(*FB_Init is always available implicitly and it is used primarily for initialization.
The return value is not evaluated. For a specific influence, you can also declare the
methods explicitly and provide additional code there with the standard initialization
code. You can evaluate the return value.*)
METHOD FB_Init : BOOL
VAR_INPUT
	(* TRUE: the retain variables are initialized (reset warm / reset cold)*)
	bInitRetains : BOOL;

	(* TRUE: the instance will be copied to the copy code afterward (online change)   *)
	bInCopyCode : BOOL;
	Name		: T_MaxString;
	Cylinder	: I_Cylinder;
END_VAR
THIS^.Cylinder := Cylinder;
Events.GenerateTcEvents(Cylinder.Name, ADR(TC_events.Cylinder), SIZEOF(ST_Cylinder));
END_METHOD

END_FUNCTION_BLOCK

// Events/Interface/I_EventReactionTcEvents
INTERFACE I_EventReactionTcEvents EXTENDS I_EventReaction

METHOD GetHighestActiveEventSeverity : TcEventSeverity
END_METHOD

END_INTERFACE

// Events/Interface/I_EventReaction
INTERFACE I_EventReaction EXTENDS I_Resettable

METHOD GetHighestActiveEventReaction : DINT;
END_METHOD

METHOD SetEventReactions
VAR_INPUT
	Verbose	 : DINT := 0;
	Info	 : DINT := 1;
	Warning	 : DINT := 2;
	Error	 : DINT := 3;
	Critical : DINT := 4;
END_VAR
END_METHOD

END_INTERFACE

// Events/TcEventClass
{attribute 'enable_dynamic_creation'}
FUNCTION_BLOCK TcEventClass EXTENDS CyclicComponent IMPLEMENTS I_EventClassTcEvents
VAR
	pEventClass				   : PVOID;
	pEventBuffer			   : POINTER TO PVOID;
	pEventTriggerBuffer		   : POINTER TO PVOID;
	pEventAutoResetBuffer	   : POINTER TO PVOID;
	NullEvent				   : FB_TcAlarm;
	NullBool				   : BOOL;
	NumberOfEvents			   : UDINT;
	HighestActiveEventSeverity : TcEventSeverity;
	EventReactionVerbose	   : DINT := 0;
	EventReactionInfo		   : DINT := 1;
	EventReactionWarning	   : DINT := 2;
	EventReactionError		   : DINT := 3;
	EventReactionCritical	   : DINT := 4;
	TcEventClassArguments	   : TcEventClassArguments;
END_VAR

METHOD Dispose
VAR
	i				: UDINT;
	pEvent			: POINTER TO FB_TcAlarm;
	pDispose		: POINTER TO TcEventClass;
	pEventAutoReset : POINTER TO BOOL;
END_VAR
pDispose := THIS;
FOR i := 1 TO NumberOfEvents DO
	pEvent := GetEventInstance(i);
	__DELETE(pEvent);
	pEventAutoReset := GetEventAutoResetInstance(i);
	__DELETE(pEventAutoReset);
END_FOR

__DELETE(pEventBuffer);
__DELETE(pDispose);
__DELETE(pEventTriggerBuffer);
__DELETE(pEventAutoResetBuffer);
END_METHOD

//FB_Exit must be implemented explicitly. If there is an implementation, then the

//method is called before the controller removes the code of the function block instance

//(implicit call). The return value is not evaluated.
METHOD FB_Exit : BOOL
VAR_INPUT
	bInCopyCode : BOOL; // TRUE: the exit method is called in order to leave the instance which will be copied afterwards (online change).  
END_VAR

VAR
	i				: UDINT;
	pEvent			: POINTER TO FB_TcAlarm;
	pEventAutoReset : POINTER TO BOOL;
END_VAR
FOR i := 1 TO NumberOfEvents DO
	pEvent := GetEventInstance(i);
	__DELETE(pEvent);
	pEventAutoReset := GetEventAutoResetInstance(i);
	__DELETE(pEventAutoReset);
END_FOR

__DELETE(pEventBuffer);
__DELETE(pEventTriggerBuffer);
__DELETE(pEventAutoResetBuffer);
END_METHOD

METHOD ClearEventById
VAR_INPUT
	EventId : UDINT;
END_VAR

VAR
	pEvent : POINTER TO FB_TcAlarm;
END_VAR
IF CheckEventId(EventId) THEN
	pEvent := GetEventInstance(EventId);
	IF (pEvent <> 0) THEN
		IF pEvent^.bRaised THEN
			pEvent^.Clear();
			FindActiveSeverity();
		END_IF
	END_IF
END_IF
END_METHOD

METHOD GetHighestActiveEventReaction : DINT
CASE HighestActiveEventSeverity OF
	TcEventSeverity.Verbose:
		GetHighestActiveEventReaction := EventReactionVerbose;

	TcEventSeverity.Info:
		GetHighestActiveEventReaction := EventReactionInfo;

	TcEventSeverity.Warning:
		GetHighestActiveEventReaction := EventReactionWarning;

	TcEventSeverity.Error:
		GetHighestActiveEventReaction := EventReactionError;

	TcEventSeverity.Critical:
		GetHighestActiveEventReaction := EventReactionCritical;
END_CASE
END_METHOD

METHOD GetHighestActiveEventSeverity : TcEventSeverity
GetHighestActiveEventSeverity := HighestActiveEventSeverity;
END_METHOD

{attribute 'monitoring' := 'call'}
PROPERTY IsResettable : BOOL
GET
VAR
	i		  : UDINT;
	pEvent	  : POINTER TO FB_TcAlarm;
	pTrigger  : POINTER TO BOOL;
END_VAR
IsResettable := FALSE;
FOR i := 1 TO NumberOfEvents DO
	pTrigger := GetEventTriggerInstance(i);
	IF (pTrigger <> 0) THEN
		pEvent := GetEventInstance(i);
		IF (pEvent <> 0) AND_THEN NOT pTrigger^ AND pEvent^.bRaised THEN
			IsResettable := TRUE;
		END_IF
	END_IF
END_FOR
END_GET
END_PROPERTY

METHOD RaiseEvent
VAR_INPUT
	EventId	  : UDINT;
END_VAR

VAR
	pEvent : POINTER TO FB_TcAlarm;
END_VAR
IF CheckEventId(EventId) THEN
	pEvent := GetEventInstance(EventId);
	IF (pEvent <> 0) THEN
		IF NOT pEvent^.bRaised THEN
			pEvent^.Raise();
			IF pEvent^.eSeverity > HighestActiveEventSeverity THEN
				HighestActiveEventSeverity := pEvent^.eSeverity;
			END_IF

			pEvent^.ipArguments.Clear();
		END_IF
	END_IF
END_IF
END_METHOD

METHOD ResetBySeverity : BOOL
VAR_INPUT
	Severity : UDINT;
END_VAR

VAR
	i	   : UDINT;
	pEvent : POINTER TO FB_TcAlarm;
END_VAR
FOR i := 1 TO NumberOfEvents DO
	pEvent := GetEventInstance(i);
	IF (pEvent <> 0) AND_THEN (pEvent^.eSeverity <= TO_DINT(Severity)) THEN
		pEvent^.Clear();
	END_IF
END_FOR

FindActiveSeverity();
ResetBySeverity := TRUE;
END_METHOD

METHOD SetEvent
VAR_INPUT
	EventId	  : UDINT;
	Trigger	  : POINTER TO BOOL;
	AutoReset : BOOL;
END_VAR

VAR
	pBool : POINTER TO BOOL;
END_VAR
IF CheckEventId(EventId) THEN
	IF Trigger <> 0 THEN
		SetEventTriggerInstance(EventId, Trigger);
	END_IF

	pBool  := GetEventAutoResetInstance(EventId);
	pBool^ := AutoReset;
END_IF
END_METHOD

METHOD SetEventReactions
VAR_INPUT
	Verbose	 : DINT := 0;
	Info	 : DINT := 1;
	Warning	 : DINT := 2;
	Error	 : DINT := 3;
	Critical : DINT := 4;
END_VAR
EventReactionVerbose  := Verbose;
EventReactionInfo	  := Info;
EventReactionWarning  := Warning;
EventReactionError	  := Error;
EventReactionCritical := Critical;
END_METHOD

METHOD PROTECTED CheckEventId : BOOL
VAR_INPUT
	EventId : UDINT;
END_VAR
CheckEventId := (EventID > 0) AND (EventId <= NumberOfEvents) AND (pEventBuffer <> 0);
END_METHOD

METHOD PROTECTED FindActiveSeverity
VAR
	i	   : UDINT;
	pEvent : POINTER TO FB_TcAlarm;
END_VAR
HighestActiveEventSeverity := Global.TcEventSeverity.Verbose;
FOR i := 1 TO NumberOfEvents DO
	pEvent := GetEventInstance(i);
	IF (pEvent <> 0) AND_THEN pEvent^.bRaised AND_THEN pEvent^.eSeverity > HighestActiveEventSeverity THEN
		HighestActiveEventSeverity := pEvent^.eSeverity;
	END_IF
END_FOR
END_METHOD

METHOD PROTECTED GetEventAutoResetInstance : POINTER TO BOOL
VAR_INPUT
	EventId : UDINT;
END_VAR

VAR
	ppEventAutoReset : POINTER TO POINTER TO BOOL;
END_VAR
IF CheckEventId(EventId) THEN
	ppEventAutoReset := pEventAutoResetBuffer + ((EventId - 1) * SIZEOF(PVOID));
	GetEventAutoResetInstance := ppEventAutoReset^;
ELSE
	GetEventAutoResetInstance := ADR(NullBool);
END_IF
END_METHOD

METHOD PROTECTED GetEventInstance : POINTER TO FB_TcAlarm
VAR_INPUT
	EventId : UDINT;
END_VAR

VAR
	ppEvent : POINTER TO POINTER TO FB_TcAlarm;
END_VAR
IF CheckEventId(EventId) THEN
	ppEvent			 := pEventBuffer + ((EventId - 1) * SIZEOF(PVOID));
	GetEventInstance := ppEvent^;
ELSE
	GetEventInstance := ADR(NullEvent);
END_IF
END_METHOD

METHOD PROTECTED GetEventTriggerInstance : POINTER TO BOOL
VAR_INPUT
	EventId : UDINT;
END_VAR

VAR
	ppEventTrigger : POINTER TO POINTER TO BOOL;
END_VAR
IF CheckEventId(EventId) THEN
	ppEventTrigger := pEventTriggerBuffer + ((EventId - 1) * SIZEOF(PVOID));
	GetEventTriggerInstance := ppEventTrigger^;
ELSE
	GetEventTriggerInstance := ADR(NullBool);
END_IF
END_METHOD

METHOD PROTECTED SetEventTriggerInstance
VAR_INPUT
	EventId : UDINT;
    Trigger : POINTER TO BOOL;
END_VAR

VAR
	ppEventTrigger : POINTER TO POINTER TO BOOL;
END_VAR
IF CheckEventId(EventId) THEN
	ppEventTrigger	:= pEventTriggerBuffer + ((EventId - 1) * SIZEOF(PVOID));
	ppEventTrigger^ := Trigger;
END_IF
END_METHOD

METHOD Reset
VAR
	i		 : UDINT;
	pEvent	 : POINTER TO FB_TcAlarm;
	pTrigger : POINTER TO BOOL;
END_VAR
FOR i := 1 TO NumberOfEvents DO
	pTrigger := GetEventTriggerInstance(i);
	pEvent	 := GetEventInstance(i);
	IF (pEvent <> 0) THEN
		IF (pTrigger <> 0) AND_THEN NOT pTrigger^ THEN
			pEvent^.Clear();
		END_IF

		IF (pTrigger = 0) THEN
			pEvent^.Clear();
		END_IF
	END_IF
END_FOR

HighestActiveEventSeverity := Global.TcEventSeverity.Verbose;
END_METHOD

METHOD PUBLIC Arguments : I_EventArguments
VAR_INPUT
	EventId : UDINT;
END_VAR

VAR
	pEvent : POINTER TO FB_TcAlarm;
END_VAR
IF CheckEventId(EventId) THEN
	pEvent := GetEventInstance(EventId);
	IF (pEvent <> 0) THEN
		TcEventClassArguments.Event := pEvent;
	ELSE
		TcEventClassArguments.Event := ADR(NullEvent);
	END_IF
ELSE
	TcEventClassArguments.Event := ADR(NullEvent);
END_IF

Arguments := TcEventClassArguments;
END_METHOD

METHOD CyclicLogic
VAR
	i	   : UDINT;
	pEvent : POINTER TO FB_TcAlarm;
	pTrigger  : POINTER TO BOOL;
    AutoReset : BOOL;
END_VAR
FOR i := 1 TO NumberOfEvents DO
	pTrigger := GetEventTriggerInstance(i);
	IF (pTrigger <> 0) THEN
		pEvent	  := GetEventInstance(i);
		AutoReset := GetEventAutoResetInstance(i)^;
		IF (pEvent <> 0) AND_THEN AutoReset AND NOT pTrigger^ THEN
			pEvent^.Clear();
			FindActiveSeverity();
		END_IF

		IF (pEvent <> 0) AND_THEN pTrigger^ THEN
			pEvent^.Raise(0);
			FindActiveSeverity();
		END_IF
	END_IF
END_FOR
END_METHOD

METHOD PUBLIC GenerateTcEvents
VAR_INPUT
	Name   : T_MaxString;
	pClass : PVOID; // ADR(TC_Events.XY) - TC Event Class in TypeSystem
	nSize  : UDINT; // SIZEOF(ST_XY) - TC Event Class in TypeSystem
END_VAR

VAR
	i				 : UDINT;
	pEventDef		 : POINTER TO TcEventEntry;
	pEvent			 : POINTER TO FB_TcAlarm;
	pBuffer			 : PVOID;
	ppBuffer		 : POINTER TO POINTER TO FB_TcAlarm;
	SourceInfo		 : FB_TcSourceInfo;
	pEventAutoReset	 : POINTER TO BOOL;
	ppEventAutoReset : POINTER TO POINTER TO BOOL;
END_VAR
NumberOfEvents		  := nSize / SIZEOF(TcEventEntry);
pEventBuffer		  := __NEW(PVOID, NumberOfEvents);
pEventTriggerBuffer	  := __NEW(PVOID, NumberOfEvents);
pEventAutoResetBuffer := __NEW(PVOID, NumberOfEvents);
pEventClass			  := pClass;
IF pEventBuffer <> 0 THEN
	SourceInfo.ResetToDefault();
	SourceInfo.sName := Name;
	FOR i := 1 TO NumberOfEvents DO
		pEvent	  := __NEW(FB_TcAlarm);
		ppBuffer  := pEventBuffer + ((i - 1) * SIZEOF(PVOID));
		ppBuffer^ := pEvent;
		pEventDef := pEventClass + ((i - 1) * SIZEOF(TcEventEntry));
		pEvent^.CreateEx2(pEventDef^, SourceInfo);

		//
		pEventAutoReset	  := __NEW(BOOL);
		ppEventAutoReset  := pEventAutoResetBuffer + ((i - 1) * SIZEOF(PVOID));
		ppEventAutoReset^ := pEventAutoReset;
	END_FOR
END_IF
END_METHOD

END_FUNCTION_BLOCK

// Events/Interface/I_EventClassTcEvents
INTERFACE I_EventClassTcEvents EXTENDS I_EventClass

METHOD PUBLIC GenerateTcEvents
VAR_INPUT
	Name   : T_MaxString;
	pClass : PVOID; // ADR(TC_Events.XY) - TC Event Class in TypeSystem
	nSize  : UDINT; // SIZEOF(ST_XY) - TC Event Class in TypeSystem
END_VAR
END_METHOD

METHOD GetHighestActiveEventSeverity : TcEventSeverity
END_METHOD

END_INTERFACE

// Events/Interface/I_EventClass
INTERFACE I_EventClass EXTENDS I_EventReaction, I_Resettable

METHOD PUBLIC Arguments : I_EventArguments
VAR_INPUT
	EventId : UDINT;
END_VAR
END_METHOD

METHOD PUBLIC ClearEventById
VAR_INPUT
	EventId : UDINT;
END_VAR
END_METHOD

{attribute 'monitoring' := 'call'}
PROPERTY IsResettable : BOOL
GET
END_GET
END_PROPERTY

METHOD PUBLIC RaiseEvent
VAR_INPUT
	EventId	  : UDINT;
END_VAR
END_METHOD

METHOD ResetBySeverity : BOOL
VAR_INPUT
	Severity : UDINT;
END_VAR
END_METHOD

METHOD SetEvent
VAR_INPUT
	EventId	  : UDINT;
	Trigger	  : POINTER TO BOOL;
	AutoReset : BOOL;
END_VAR
END_METHOD

END_INTERFACE

// Components/Digital/Visitor/ForceVisitor
FUNCTION_BLOCK ForceVisitor IMPLEMENTS I_ComponentVisitor
VAR
	Forcible : I_ForcibleBool;
	{attribute 'hide'}
	_ForceState : E_ForceState;
END_VAR

{attribute 'monitoring' := 'call'}
PROPERTY Force : E_ForceState
GET
Force := _ForceState;
END_GET
SET
_ForceState := Force;
END_SET
END_PROPERTY

METHOD VisitComponent
VAR_INPUT
	Component : I_Component;
END_VAR
IF __QUERYINTERFACE(Component, Forcible) THEN
	Forcible.Force := Force;
END_IF
END_METHOD

END_FUNCTION_BLOCK

// Components/Digital/Visitor/ReleaseAllForceVisitor
FUNCTION_BLOCK ReleaseAllForceVisitor IMPLEMENTS I_ModuleVisitor, I_ComponentVisitor
VAR
END_VAR

METHOD ReleaseForces : BOOL;
VAR_INPUT
	Module : I_Module;
END_VAR
Module.Accept(THIS^);
END_METHOD

METHOD VisitComponent
VAR_INPUT
	Component : I_Component;
END_VAR

VAR_INST
	Forcible : I_ForcibleBool;
END_VAR
IF __QUERYINTERFACE(Component, Forcible) THEN
	Forcible.Force := E_ForceState.Unforced;
END_IF
END_METHOD

METHOD VisitModule
VAR_INPUT
	Module : I_Module;
END_VAR
Module.Components.Accept(THIS^);
Module.Modules.Accept(THIS^);
END_METHOD

END_FUNCTION_BLOCK

// Components/Digital/DigitalInput_Combiner
FUNCTION_BLOCK DigitalInput_Combiner
VAR_GENERIC CONSTANT
	NumberOfCombinedInputs : DINT := 2;
END_VAR
EXTENDS Component IMPLEMENTS I_DigitalInput
VAR
	Inputs : ARRAY[0..(NumberOfCombinedInputs - 1)] OF I_DigitalInput;
	{attribute 'hide'}
	_Force : E_ForceState;
END_VAR

METHOD AddInput
VAR_INPUT
	Input : I_DigitalInput;
END_VAR

VAR
	i : DINT;
END_VAR
FOR i := 0 TO (NumberOfCombinedInputs - 1) DO
	IF Inputs[i] = Input THEN
		RETURN;
	END_IF
END_FOR

FOR i := 0 TO (NumberOfCombinedInputs - 1) DO
	IF Inputs[i] = 0 THEN
		Inputs[i] := Input;
		RETURN;
	END_IF
END_FOR
END_METHOD

{attribute 'monitoring' := 'call'}
PROPERTY Force : E_ForceState
GET
Force := _Force;
END_GET
SET
VAR
	i : DINT;
END_VAR
_Force := Force;
IF Inputs[0] = 0 THEN
	RETURN;
END_IF

FOR i := 0 TO (NumberOfCombinedInputs - 1) DO
	IF Inputs[i] = 0 THEN
		RETURN;
	END_IF

	Inputs[i].Force := Force;
END_FOR
END_SET
END_PROPERTY

{attribute 'monitoring' := 'call'}
PROPERTY IsActive : BOOL
GET
VAR
	i : DINT;
END_VAR
IF Inputs[0] = 0 THEN
	RETURN;
END_IF

IsActive := TRUE;
FOR i := 0 TO (NumberOfCombinedInputs - 1) DO
	IF Inputs[i] = 0 THEN
		RETURN;
	END_IF

	IsActive := IsActive AND Inputs[i].IsActive;
END_FOR
END_GET
END_PROPERTY

END_FUNCTION_BLOCK

// Components/Digital/DigitalInput_DebounceFallingEdge
FUNCTION_BLOCK DigitalInput_DebounceFallingEdge EXTENDS CyclicComponent IMPLEMENTS I_DigitalInput
VAR
	Input : I_DigitalInput;
	{attribute 'hide'}
	_DebounceTime		: TIME;
	DebounceFallingEdge : TOF;
END_VAR

METHOD CyclicLogic
DebounceFallingEdge(IN := Input.IsActive, PT := _DebounceTime);
END_METHOD

{attribute 'monitoring' := 'call'}
PROPERTY DebounceTime : TIME
GET
DebounceTime := _DebounceTime;
END_GET
SET
_DebounceTime := DebounceTime;
END_SET
END_PROPERTY

(*FB_Init is always available implicitly and it is used primarily for initialization.
The return value is not evaluated. For a specific influence, you can also declare the
methods explicitly and provide additional code there with the standard initialization
code. You can evaluate the return value.*)
METHOD FB_Init : BOOL
VAR_INPUT
	(* TRUE: the retain variables are initialized (reset warm / reset cold)*)
	bInitRetains : BOOL;

	(* TRUE: the instance will be copied to the copy code afterward (online change)   *)
	bInCopyCode : BOOL;
	Name		: T_MaxString;
	Input		: I_DigitalInput;
END_VAR
THIS^.Input := Input;
END_METHOD

{attribute 'monitoring' := 'call'}
PROPERTY Force : E_ForceState
GET
Force := Input.Force;
END_GET
SET
Input.Force := Force;
END_SET
END_PROPERTY

{attribute 'monitoring' := 'call'}
PROPERTY IsActive : BOOL
GET
IsActive := DebounceFallingEdge.Q;
END_GET
END_PROPERTY

END_FUNCTION_BLOCK

// Components/Digital/DigitalInput_DebounceRisingEdge
FUNCTION_BLOCK DigitalInput_DebounceRisingEdge EXTENDS CyclicComponent IMPLEMENTS I_DigitalInput
VAR
	Input : I_DigitalInput;
	{attribute 'hide'}
	_DebounceTime	   : TIME;
	DebounceRisingEdge : TON;
END_VAR

METHOD CyclicLogic
DebounceRisingEdge(IN := Input.IsActive, PT := _DebounceTime);
END_METHOD

{attribute 'monitoring' := 'call'}
PROPERTY DebounceTime : TIME
GET
DebounceTime := _DebounceTime;
END_GET
SET
_DebounceTime := DebounceTime;
END_SET
END_PROPERTY

(*FB_Init is always available implicitly and it is used primarily for initialization.
The return value is not evaluated. For a specific influence, you can also declare the
methods explicitly and provide additional code there with the standard initialization
code. You can evaluate the return value.*)
METHOD FB_Init : BOOL
VAR_INPUT
	(* TRUE: the retain variables are initialized (reset warm / reset cold)*)
	bInitRetains : BOOL;

	(* TRUE: the instance will be copied to the copy code afterward (online change)   *)
	bInCopyCode : BOOL;
	Name		: T_MaxString;
	Input		: I_DigitalInput;
END_VAR
THIS^.Input := Input;
END_METHOD

{attribute 'monitoring' := 'call'}
PROPERTY Force : E_ForceState
GET
Force := Input.Force;
END_GET
SET
Input.Force := Force;
END_SET
END_PROPERTY

{attribute 'monitoring' := 'call'}
PROPERTY IsActive : BOOL
GET
IsActive := DebounceRisingEdge.Q;
END_GET
END_PROPERTY

END_FUNCTION_BLOCK

// Components/Digital/DigitalInput_HMI
FUNCTION_BLOCK DigitalInput_HMI EXTENDS HmiFunction
VAR
	DigitalInput : I_DigitalInput;
	{ attribute 'TcHmiSymbol.AddSymbol' }
	{ attribute 'TcHmiSymbol.AddSymbol.UserGroups' := '__SystemAdministrators,Admin' }
	DigitalInput_HMI : ST_DigitalInput_HMI;
END_VAR

PROPERTY ControlObject : I_Base
SET
__QueryInterface(ControlObject,DigitalInput);
END_SET
END_PROPERTY

METHOD CyclicLogic
IF DigitalInput = 0 THEN
	RETURN;
END_IF

DigitalInput_HMI.Name		:= DigitalInput.Name;
DigitalInput_HMI.Active		:= DigitalInput.IsActive;
DigitalInput_HMI.HmiEnabled := Enabled;
IF Enabled THEN
	DigitalInput.Force := DigitalInput_HMI.Force;
END_IF
END_METHOD

(*FB_Init is always available implicitly and it is used primarily for initialization.
The return value is not evaluated. For a specific influence, you can also declare the
methods explicitly and provide additional code there with the standard initialization
code. You can evaluate the return value.*)
METHOD FB_Init : BOOL
VAR_INPUT
	(* TRUE: the retain variables are initialized (reset warm / reset cold)*)
	bInitRetains : BOOL;

	(* TRUE: the instance will be copied to the copy code afterward (online change)   *)
	bInCopyCode	 : BOOL;
	Name		 : T_MaxString;
	DigitalInput : I_DigitalInput;
END_VAR
THIS^.DigitalInput := DigitalInput;
ControlType		   := 'DigitalInput';
LinkObject		   := 'DigitalInput_HMI';
END_METHOD

END_FUNCTION_BLOCK

// Components/Digital/DigitalInput_NC
FUNCTION_BLOCK DigitalInput_NC EXTENDS Component IMPLEMENTS I_DigitalInput
VAR
	Input		  : REFERENCE TO BOOL;
	ForcibleInput : ForcibleBool(_Name);
END_VAR

//FB_Init is always available implicitly and it is used primarily for initialization.

//The return value is not evaluated. For a specific influence, you can also declare the

//methods explicitly and provide additional code there with the standard initialization

//code. You can evaluate the return value.
METHOD FB_Init : BOOL
VAR_INPUT
	bInitRetains : BOOL; // TRUE: the retain variables are initialized (reset warm / reset cold)
	bInCopyCode	 : BOOL; // TRUE: the instance will be copied to the copy code afterward (online change)   
	Name		 : T_MaxString;
	Input		 : REFERENCE TO BOOL;
END_VAR
THIS^.Input REF= Input;
END_METHOD

{attribute 'monitoring' := 'call'}
PROPERTY Force : E_ForceState
GET
Force := ForcibleInput.CurrentForceState;
END_GET
SET
VAR
	ForceString : T_MaxString := TO_STRING(Force);
END_VAR
ForcibleInput.SetForceState(Force);
END_SET
END_PROPERTY

{attribute 'monitoring' := 'call'}
PROPERTY IsActive : BOOL
GET
ForcibleInput.Input := NOT Input;
IsActive			:= ForcibleInput.Output;
END_GET
END_PROPERTY

END_FUNCTION_BLOCK

// Components/Digital/DigitalOutput_HMI
FUNCTION_BLOCK DigitalOutput_HMI EXTENDS HmiFunction
VAR
	DigitalOutput : I_DigitalOutput;
	{ attribute 'TcHmiSymbol.AddSymbol' }
	{ attribute 'TcHmiSymbol.AddSymbol.UserGroups' := '__SystemAdministrators,Admin' }
	DigitalOutput_HMI : ST_DigitalOutput_HMI;
END_VAR

PROPERTY ControlObject : I_Base
SET
__QueryInterface(ControlObject,DigitalOutput);
END_SET
END_PROPERTY

METHOD CyclicLogic
IF DigitalOutput = 0 THEN
	RETURN;
END_IF

DigitalOutput_HMI.Name		 := DigitalOutput.Name;
DigitalOutput_HMI.On		 := DigitalOutput.On;
DigitalOutput_HMI.HmiEnabled := Enabled;
IF Enabled THEN
	DigitalOutput.Force := DigitalOutput_HMI.Force;
END_IF
END_METHOD

(*FB_Init is always available implicitly and it is used primarily for initialization.
The return value is not evaluated. For a specific influence, you can also declare the
methods explicitly and provide additional code there with the standard initialization
code. You can evaluate the return value.*)
METHOD FB_Init : BOOL
VAR_INPUT
	(* TRUE: the retain variables are initialized (reset warm / reset cold)*)
	bInitRetains : BOOL;

	(* TRUE: the instance will be copied to the copy code afterward (online change)   *)
	bInCopyCode	  : BOOL;
	Name		  : T_MaxString;
	DigitalOutput : I_DigitalOutput;
END_VAR
THIS^.DigitalOutput := DigitalOutput;
ControlType			:= 'DigitalOutput';
LinkObject			:= 'DigitalOutput_HMI';
END_METHOD

END_FUNCTION_BLOCK

// Components/EtherCat/Interface/I_EcIoDevice
INTERFACE I_EcIoDevice EXTENDS I_IoDevice, I_CoeAccess

{attribute 'monitoring' := 'call'}
PROPERTY Bootstrap : BOOL
GET
END_GET
END_PROPERTY

PROPERTY Configuration : REFERENCE TO ST_EcSlaveConfigData
GET
END_GET
SET
END_SET
END_PROPERTY

{attribute 'monitoring' := 'call'}
PROPERTY DeviceError : BOOL
GET
END_GET
END_PROPERTY

{attribute 'monitoring' := 'call'}
PROPERTY Disabled : BOOL
GET
END_GET
END_PROPERTY

{attribute 'monitoring' := 'call'}
PROPERTY Init : BOOL
GET
END_GET
END_PROPERTY

{attribute 'monitoring' := 'call'}
PROPERTY InitCmdError : BOOL
GET
END_GET
END_PROPERTY

{attribute 'monitoring' := 'call'}
PROPERTY InvalidVPRS : BOOL
GET
END_GET
END_PROPERTY

{attribute 'monitoring' := 'call'}
PROPERTY OP : BOOL
GET
END_GET
END_PROPERTY

{attribute 'monitoring' := 'call'}
PROPERTY PreOp : BOOL
GET
END_GET
END_PROPERTY

{attribute 'monitoring' := 'call'}
PROPERTY SafeOp : BOOL
GET
END_GET
END_PROPERTY

PROPERTY State : REFERENCE TO ST_EcSlaveState
GET
END_GET
SET
END_SET
END_PROPERTY

END_INTERFACE

// Components/EtherCat/Interface/I_IoDevice
INTERFACE I_IoDevice EXTENDS I_Base

{attribute 'monitoring' := 'call'}
PROPERTY IoDataValid : BOOL
GET
END_GET
END_PROPERTY

END_INTERFACE

// Components/EtherCat/Interface/I_EtherCatDiagnosticEventProvider
INTERFACE I_EtherCatDiagnosticEventProvider EXTENDS I_EventReactionTcEvents

METHOD RaiseEtherCatDiagnosticEvent
VAR_INPUT
	EventId	  : UDINT;
	Argument1 : STRING := '';
	Argument2 : STRING := '';
	Argument3 : STRING := '';
END_VAR
END_METHOD

METHOD RaiseSyncUnitEvent
VAR_INPUT
	EventId	  : UDINT;
	Argument1 : STRING := '';
	Argument2 : STRING := '';
	Argument3 : STRING := '';
END_VAR
END_METHOD

END_INTERFACE

// Components/EtherCat/Interface/I_EtherCatMasterDiagnostic
INTERFACE I_EtherCatMasterDiagnostic EXTENDS I_Component, I_Resettable

{attribute 'monitoring' := 'call'}
PROPERTY ConfiguredSlaveCount : UINT
GET
END_GET
END_PROPERTY

METHOD GetIoDeviceByAddr : I_EcIoDevice
VAR_INPUT
	Addr : WORD;
END_VAR
END_METHOD

METHOD GetIoDeviceByName : I_EcIoDevice
VAR_INPUT
	Name : STRING(31);
END_VAR
END_METHOD

{attribute 'monitoring' := 'call'}
PROPERTY LocalAmsNetId : T_AmsNetId
GET
END_GET
END_PROPERTY

{attribute 'monitoring' := 'call'}
PROPERTY MasterAmsNetId : T_AmsNetId
GET
END_GET
END_PROPERTY

METHOD RegisterEventProvider
VAR_INPUT
	EventProvider : I_EtherCatDiagnosticEventProvider;
END_VAR
END_METHOD

{attribute 'monitoring' := 'call'}
PROPERTY SlaveCount : UINT
GET
END_GET
END_PROPERTY

END_INTERFACE

// Components/EtherCat/Interface/I_SyncUnitTask
INTERFACE I_SyncUnitTask EXTENDS I_Component

{attribute 'monitoring' := 'call'}
PROPERTY IoDataValid : BOOL
GET
END_GET
END_PROPERTY

{attribute 'monitoring' := 'call'}
PROPERTY IsHotConnect : BOOL
GET
END_GET
END_PROPERTY

{attribute 'monitoring' := 'call'}
PROPERTY PUBLIC SlaveCount : UINT
GET
END_GET
END_PROPERTY

END_INTERFACE

// Components/EtherCat/EtherCatIoDevice
FUNCTION_BLOCK EtherCatIoDevice EXTENDS CyclicComponent IMPLEMENTS I_EcIoDevice
VAR
	_Config	  : REFERENCE TO ST_EcSlaveConfigData;
	_State	  : REFERENCE TO ST_EcSlaveState;
	_SyncUnit : I_SyncUnitTask;
	_AmsAddr  : AMSADDR;
	CoeDevice : CoeDevice('CoE Terminal');
	{attribute 'hide'}
	NullCoeDevice : NullCoeDevice('Null Terminal');
END_VAR

{attribute 'monitoring' := 'call'}
PROPERTY Bootstrap : BOOL
GET
VAR
	DiagByte	: BYTE;
	BitMaskDiag : BYTE := 16#0F;
END_VAR
IF __ISVALIDREF(_State) THEN
	BitMaskDiag := 16#0F;
	DiagByte	:= _State.deviceState AND BitMaskDiag;
	Bootstrap	:= DiagByte = EC_DEVICE_STATE_BOOTSTRAP;
END_IF
END_GET
END_PROPERTY

PROPERTY CoE : I_CoeDevice
GET
IF _Config.nMailboxInSize = 0 THEN
	CoE := NullCoeDevice;
ELSE
	_AmsAddr.port	  := _Config.nAddr;
	CoeDevice.AdsAddr REF= _AmsAddr;
	CoE				  := CoeDevice;
END_IF
END_GET
SET
END_SET
END_PROPERTY

PROPERTY Configuration : REFERENCE TO ST_EcSlaveConfigData
GET
Configuration REF= _Config;
END_GET
SET
_Config REF= Configuration;
END_SET
END_PROPERTY

{attribute 'monitoring' := 'call'}
PROPERTY DeviceError : BOOL
GET
VAR
	DiagByte	: BYTE;
	BitMaskDiag : BYTE := 16#0F;
END_VAR
IF __ISVALIDREF(_State) THEN
	BitMaskDiag := 16#0F;
	DiagByte	:= _State.deviceState AND BitMaskDiag;
	DeviceError := DiagByte = EC_DEVICE_STATE_ERROR;
END_IF
END_GET
END_PROPERTY

{attribute 'monitoring' := 'call'}
PROPERTY Disabled : BOOL
GET
VAR
	DiagByte	: BYTE;
	BitMaskDiag : BYTE := 16#0F;
END_VAR
IF __ISVALIDREF(_State) THEN
	BitMaskDiag := 16#0F;
	DiagByte	:= _State.deviceState AND BitMaskDiag;
	Disabled	:= DiagByte = EC_DEVICE_STATE_DISABLED;
END_IF
END_GET
END_PROPERTY

{attribute 'monitoring' := 'call'}
PROPERTY Init : BOOL
GET
VAR
	DiagByte	: BYTE;
	BitMaskDiag : BYTE := 16#0F;
END_VAR
IF __ISVALIDREF(_State) THEN
	BitMaskDiag := 16#0F;
	DiagByte	:= _State.deviceState AND BitMaskDiag;
	Init		:= DiagByte = EC_DEVICE_STATE_INIT;
END_IF
END_GET
END_PROPERTY

{attribute 'monitoring' := 'call'}
PROPERTY InitCmdError : BOOL
GET
VAR
	DiagByte	: BYTE;
	BitMaskDiag : BYTE := 16#0F;
END_VAR
IF __ISVALIDREF(_State) THEN
	BitMaskDiag	 := 16#0F;
	DiagByte	 := _State.deviceState AND BitMaskDiag;
	InitCmdError := DiagByte = EC_DEVICE_STATE_INVALID_VPRS;
END_IF
END_GET
END_PROPERTY

{attribute 'monitoring' := 'call'}
PROPERTY InvalidVPRS : BOOL
GET
VAR
	DiagByte	: BYTE;
	BitMaskDiag : BYTE := 16#0F;
END_VAR
IF __ISVALIDREF(_State) THEN
	BitMaskDiag := 16#0F;
	DiagByte	:= _State.deviceState AND BitMaskDiag;
	InvalidVPRS := DiagByte = EC_DEVICE_STATE_INVALID_VPRS;
END_IF
END_GET
END_PROPERTY

{attribute 'monitoring' := 'call'}
PROPERTY IoDataValid : BOOL
GET
IF _SyncUnit <> 0 THEN
	IoDataValid := _SyncUnit.IoDataValid;
ELSE
	IoDataValid := TRUE;
END_IF
END_GET
END_PROPERTY

{attribute 'monitoring' := 'call'}
PROPERTY OP : BOOL
GET
VAR
	DiagByte	: BYTE;
	BitMaskDiag : BYTE := 16#0F;
END_VAR
IF __ISVALIDREF(_State) THEN
	BitMaskDiag := 16#0F;
	DiagByte	:= _State.deviceState AND BitMaskDiag;
	OP			:= DiagByte = EC_DEVICE_STATE_OP;
END_IF
END_GET
END_PROPERTY

{attribute 'monitoring' := 'call'}
PROPERTY PreOp : BOOL
GET
VAR
	DiagByte	: BYTE;
	BitMaskDiag : BYTE := 16#0F;
END_VAR
IF __ISVALIDREF(_State) THEN
	BitMaskDiag := 16#0F;
	DiagByte	:= _State.deviceState AND BitMaskDiag;
	PreOp		:= DiagByte = EC_DEVICE_STATE_PREOP;
END_IF
END_GET
END_PROPERTY

{attribute 'monitoring' := 'call'}
PROPERTY SafeOp : BOOL
GET
VAR
	DiagByte	: BYTE;
	BitMaskDiag : BYTE := 16#0F;
END_VAR
IF __ISVALIDREF(_State) THEN
	BitMaskDiag := 16#0F;
	DiagByte	:= _State.deviceState AND BitMaskDiag;
	SafeOp		:= DiagByte = EC_DEVICE_STATE_SAFEOP;
END_IF
END_GET
END_PROPERTY

PROPERTY State : REFERENCE TO ST_EcSlaveState
GET
State REF= _State;
END_GET
SET
_State REF= State;
END_SET
END_PROPERTY

PROPERTY AmsNetId : AMSNETID
SET
_AmsAddr.netId := AmsNetId;
END_SET
END_PROPERTY

METHOD CyclicLogic
IF _AmsAddr.port = 0 THEN
	_AmsAddr.port	  := _Config.nAddr;
	CoeDevice.AdsAddr REF= _AmsAddr;
END_IF

IF _Config.nMailboxInSize <> 0 THEN
	CoeDevice.CyclicLogic();
END_IF
END_METHOD

PROPERTY SyncUnit : I_SyncUnitTask
SET
_SyncUnit := SyncUnit;
END_SET
END_PROPERTY

END_FUNCTION_BLOCK

// Components/EtherCat/EtherCatMaster
FUNCTION_BLOCK EtherCatMaster
VAR_GENERIC CONSTANT
	FRAMES	   : UINT := 1;
	SYNC_UNITS : UINT := 2;
END_VAR
EXTENDS CyclicComponent IMPLEMENTS I_EtherCatMasterDiagnostic, I_Initializable, I_TaskResult, I_Simulatable
VAR
	EcMaster	AT %I*	: ST_EtherCatMasterInfo;
	FrmXWcState AT %I*	: ARRAY[0..(FRAMES - 1)] OF WORD;
	ConfiguredSlaveInfo : ARRAY[0..MAX_EC_SLAVES] OF ST_EcSlaveConfigData;
	SlavesState			: ARRAY[0..MAX_EC_SLAVES] OF ST_EcSlaveState;
	SlaveTopologyInfo	: ARRAY[0..MAX_EC_SLAVES] OF ST_TopologyDataEx;
	SyncUnit			: ARRAY[0..(SYNC_UNITS - 1)] OF SyncUnitTask('Sync Unit', THIS^, ConfiguredSlaveInfo, SlaveTopologyInfo);
	IoDevice			: ARRAY[0..MAX_EC_SLAVES] OF EtherCatIoDevice('Io Device');
	EventProvider		: I_EtherCatDiagnosticEventProvider;
END_VAR

VAR
	SlaveSequence									 : UDINT;
	RunSlaveDiag, LastFramesWcStatesOk				 : BOOL;
	LastChangeCount, LastSlaveCount, LastMasterState : UINT;
	EcStartupCycles									 : UINT;
	GetConfiguredSlaves								 : FB_EcGetConfSlaves;
	GetMasterFrameCount								 : FB_EcMasterFrameCount;
	GetAllSlaveStates								 : FB_EcGetAllSlaveStates;
	GetSlaveTopologyInfo							 : FB_EcGetSlaveTopologyInfo;
END_VAR

VAR
	{attribute 'hide'}
	_Initialized : BOOL;
	{attribute 'hide'}
	_Error : BOOL;
	{attribute 'hide'}
	_Busy : BOOL;
	{attribute 'hide'}
	_ErrorId : UDINT;
	{attribute 'hide'}
	_Simulated : BOOL;
	{attribute 'hide'}
	Config : ST_EcSlaveConfigData;
	{attribute 'hide'}
	State : ST_EcSlaveState;
	{attribute 'hide'}
	NullIoDevice : EtherCatIoDevice('NullIoDevice') := (Configuration := Config, State := State);
	{attribute 'hide'}
	_LocalAmsNetId : T_AmsNetId;
	{attribute 'hide'}
	_MasterAmsNetId : T_AmsNetId;
END_VAR

METHOD PROTECTED FramesWcStatesOk : BOOL
VAR
	i : UDINT;
END_VAR
FramesWcStatesOk := TRUE;
FOR i := 0 TO (GetMasterFrameCount.nFrames - 1) DO
	IF FrmXWcState[i] <> 0 THEN
		FramesWcStatesOk := FALSE;
		EXIT;
	END_IF
END_FOR
END_METHOD

METHOD PROTECTED LookupMasterState : STRING
VAR_INPUT
	State : UINT;
END_VAR
IF State.0 THEN
	LookupMasterState := 'Link error';
ELSIF State.1 THEN
	LookupMasterState := 'I/O locked after link error (I/O reset required)';
ELSIF State.2 THEN
	LookupMasterState := 'Link error (redundancy adapter)';
ELSIF State.3 THEN
	LookupMasterState := 'Missing one frame (redundancy mode)';
ELSIF State.4 THEN
	LookupMasterState := 'Out of send resources (I/O reset required)';
ELSIF State.5 THEN
	LookupMasterState := 'Watchdog triggered';
ELSIF State.6 THEN
	LookupMasterState := 'Ethernet driver (miniport) NOT found';
ELSIF State.7 THEN
	LookupMasterState := 'I/O reset active';
ELSIF State.8 THEN
	LookupMasterState := 'At least one device in INIT state';
ELSIF State.9 THEN
	LookupMasterState := 'At least one device in PRE-OP state';
ELSIF State.10 THEN
	LookupMasterState := 'At least one device in SAFE-OP state';
ELSIF State.11 THEN
	LookupMasterState := 'At least one device indicates an error state';
ELSIF State.12 THEN
	LookupMasterState := 'DC not in sync';
ELSE
	LookupMasterState := 'State not found';
END_IF
END_METHOD

METHOD PROTECTED LookupSlaveState : STRING
VAR_INPUT
	Slave : UINT;
END_VAR

VAR_INST
	DiagByte	: BYTE;
	BitMaskDiag : BYTE := 16#0F;
END_VAR
(* State *)
BitMaskDiag := 16#0F;
DiagByte	:= SlavesState[Slave].deviceState AND BitMaskDiag;
CASE DiagByte OF
	EC_DEVICE_STATE_INIT:
		LookupSlaveState := 'Init';

	EC_DEVICE_STATE_PREOP:
		LookupSlaveState := 'Pre-op';

	EC_DEVICE_STATE_BOOTSTRAP:
		LookupSlaveState := 'Boot';

	EC_DEVICE_STATE_SAFEOP:
		LookupSlaveState := 'Safe-op';

	EC_DEVICE_STATE_OP:
		LookupSlaveState := 'OP';

ELSE
	LookupSlaveState := '';
END_CASE

(* Additional State Bits *)
IF SlavesState[Slave].deviceState.4 THEN // EC_DEVICE_STATE_ERROR
	LookupSlaveState := CONCAT(LookupSlaveState, ' - ');
	LookupSlaveState := CONCAT(LookupSlaveState, 'State machine error in the EtherCAT slave');
END_IF

IF SlavesState[Slave].deviceState.5 THEN // EC_DEVICE_STATE_INVALID_VPRS
	LookupSlaveState := CONCAT(LookupSlaveState, ' - ');
	LookupSlaveState := CONCAT(LookupSlaveState, 'Invalid vendor ID');
END_IF

IF SlavesState[Slave].deviceState.6 THEN // EC_DEVICE_STATE_INITCMD_ERROR
	LookupSlaveState := CONCAT(LookupSlaveState, ' - ');
	LookupSlaveState := CONCAT(LookupSlaveState, 'Error during sending of initialization commands');
END_IF

IF SlavesState[Slave].deviceState.7 THEN // EC_DEVICE_STATE_DISABLED
	LookupSlaveState := CONCAT(LookupSlaveState, ' - ');
	LookupSlaveState := CONCAT(LookupSlaveState, 'Slave is disabled');
END_IF

//_____________________________________________________________________________________________________

(* Link States *)
IF SlavesState[Slave].linkState.0 THEN // EC_LINK_STATE_NOT_PRESENT
	LookupSlaveState := CONCAT(LookupSlaveState, ' - ');
	LookupSlaveState := CONCAT(LookupSlaveState, 'No EtherCAT communication with the EtherCAT slave');
END_IF

IF SlavesState[Slave].linkState.1 THEN // EC_LINK_STATE_LINK_WITHOUT_COMM
	LookupSlaveState := CONCAT(LookupSlaveState, ' - ');
	LookupSlaveState := CONCAT(LookupSlaveState, 'Error AT port X');
END_IF

IF SlavesState[Slave].linkState.2 THEN // EC_LINK_STATE_MISSING_LINK
	LookupSlaveState := CONCAT(LookupSlaveState, ' - ');
	LookupSlaveState := CONCAT(LookupSlaveState, 'Missing link AT port X');
END_IF

IF SlavesState[Slave].linkState.3 THEN // EC_LINK_STATE_ADDITIONAL_LINK
	LookupSlaveState := CONCAT(LookupSlaveState, ' - ');
	LookupSlaveState := CONCAT(LookupSlaveState, 'Additional link AT port X');
END_IF

(* Additional State Bits *)
IF SlavesState[Slave].linkState.4 THEN // EC_LINK_STATE_PORT_A
	LookupSlaveState := CONCAT(LookupSlaveState, ' - ');
	LookupSlaveState := CONCAT(LookupSlaveState, 'Port 0');
END_IF

IF SlavesState[Slave].linkState.5 THEN // EC_LINK_STATE_PORT_B
	LookupSlaveState := CONCAT(LookupSlaveState, ' - ');
	LookupSlaveState := CONCAT(LookupSlaveState, 'Port 1');
END_IF

IF SlavesState[Slave].linkState.6 THEN // EC_LINK_STATE_PORT_C
	LookupSlaveState := CONCAT(LookupSlaveState, ' - ');
	LookupSlaveState := CONCAT(LookupSlaveState, 'Port 2');
END_IF

IF SlavesState[Slave].linkState.7 THEN // EC_LINK_STATE_PORT_D
	LookupSlaveState := CONCAT(LookupSlaveState, ' - ');
	LookupSlaveState := CONCAT(LookupSlaveState, 'Port 3');
END_IF
END_METHOD

METHOD PROTECTED MasterState : BOOL
VAR_INPUT
END_VAR
IF (LastMasterState <> EcMaster.DevState) AND (EcMaster.DevState <> 0) AND (EcMaster.SlaveCount < EcMaster.CfgSlaveCount) THEN
	IF EcMaster.DevState <> 0 THEN
		IF EventProvider <> 0 THEN
			EventProvider.RaiseEtherCatDiagnosticEvent(E_EtherCatMaster.MasterError, LookupMasterState(EcMaster.DevState));
		END_IF

		_Error	 := TRUE;
		_ErrorId := EcMaster.DevState;
	END_IF
END_IF
END_METHOD

METHOD PROTECTED SlaveState : BOOL
VAR_INST
	DiagByte	 : BYTE;
	BitMaskDiag	 : BYTE := 16#0F;
	FaultedSlave : UINT;
	i, j		 : UINT;
END_VAR
CASE SlaveSequence OF
	(* Wait for start *)
	0:
		GetAllSlaveStates.bExecute	  := FALSE;
		GetSlaveTopologyInfo.bExecute := FALSE;
		IF RunSlaveDiag THEN
			RunSlaveDiag := FALSE;
			NextStep(SlaveSequence);
		END_IF

	(* Update Topology*)
	10:
		GetSlaveTopologyInfo.bExecute := TRUE;
		IF GetSlaveTopologyInfo.bBusy THEN
			NextMinorStep(SlaveSequence);
		END_IF

	11:
		IF NOT GetSlaveTopologyInfo.bBusy AND NOT GetSlaveTopologyInfo.bError THEN
			NextStep(SlaveSequence);
		END_IF

		IF GetSlaveTopologyInfo.bError THEN
			SlaveSequence := 999;
		END_IF

	(* Read Slave States *)
	20:
		GetAllSlaveStates.bExecute := TRUE;
		IF GetAllSlaveStates.bBusy THEN
			NextMinorStep(SlaveSequence);
		END_IF

	21:
		IF NOT GetAllSlaveStates.bBusy AND NOT GetAllSlaveStates.bError THEN
			NextStep(SlaveSequence);
		END_IF

		IF GetAllSlaveStates.bError THEN
			SlaveSequence := 999;
		END_IF

	(* Evaluate Slave Error *)
	30:
		FOR FaultedSlave := 0 TO (EcMaster.CfgSlaveCount - 1) DO
			BitMaskDiag := 16#0F;
			DiagByte	:= SlavesState[FaultedSlave].deviceState AND BitMaskDiag;
			IF DiagByte <> EC_DEVICE_STATE_OP AND SlaveTopologyInfo[FaultedSlave].nStatusBits.4 = FALSE THEN // No error if hotconnect
				IF SlavesState[FaultedSlave].deviceState.7 THEN												 // Slave is Disabled - warning only
					IF EventProvider <> 0 THEN
						EventProvider.RaiseEtherCatDiagnosticEvent(E_EtherCatMaster.SlaveDisabled, ConfiguredSlaveInfo[FaultedSlave].sName);
					END_IF
				ELSE
					IF EventProvider <> 0 THEN
						EventProvider.RaiseEtherCatDiagnosticEvent(E_EtherCatMaster.SlaveError, ConfiguredSlaveInfo[FaultedSlave].sName, LookupSlaveState(FaultedSlave));
					END_IF

					_Error	 := TRUE;
					_ErrorId := FaultedSlave;
					EXIT;
				END_IF
			END_IF

			BitMaskDiag := 16#0F;
			DiagByte	:= SlavesState[FaultedSlave].linkState AND BitMaskDiag;
			IF DiagByte <> EC_LINK_STATE_OK AND SlaveTopologyInfo[FaultedSlave].nStatusBits.4 = FALSE THEN // Next slave is in hotconnect group, no error
				IF EventProvider <> 0 THEN
					EventProvider.RaiseEtherCatDiagnosticEvent(E_EtherCatMaster.SlaveError, ConfiguredSlaveInfo[FaultedSlave].sName, LookupSlaveState(FaultedSlave));
				END_IF

				_Error	 := TRUE;
				_ErrorId := FaultedSlave;
				EXIT;
			END_IF
		END_FOR

		NextStep(SlaveSequence);

	(* Build Slaves *)
	40:
		FOR i := 0 TO (EcMaster.CfgSlaveCount - 1) DO
			FOR j := 0 TO (SYNC_UNITS - 1) DO
				IF SyncUnit[j].IsTerminalPartOfSyncUnit(ConfiguredSlaveInfo[i].nAddr) THEN
					IoDevice[i].SyncUnit := SyncUnit[j];
				END_IF
			END_FOR
		END_FOR

		SlaveSequence := 0;

	(* Sequence Error *)
	999:
		_ErrorId	  := 999;
		SlaveSequence := 0;
END_CASE
END_METHOD

{attribute 'monitoring' := 'call'}
PROPERTY ConfiguredSlaveCount : UINT
GET
ConfiguredSlaveCount := EcMaster.CfgSlaveCount;
END_GET
END_PROPERTY

METHOD GetIoDeviceByAddr : I_EcIoDevice
VAR_INPUT
	Addr : WORD;
END_VAR

VAR
	i : UINT;
END_VAR
IF NOT Initialized THEN
	GetIoDeviceByAddr := NullIoDevice;
	RETURN;
END_IF

FOR i := 0 TO (EcMaster.CfgSlaveCount - 1) DO
	IF IoDevice[i].Configuration.nAddr = Addr THEN
		GetIoDeviceByAddr := IoDevice[i];
		RETURN;
	END_IF
END_FOR

GetIoDeviceByAddr := NullIoDevice;
END_METHOD

METHOD GetIoDeviceByName : I_EcIoDevice
VAR_INPUT
	Name : STRING(31);
END_VAR

VAR
	i : UINT;
END_VAR
IF NOT Initialized THEN
	GetIoDeviceByName := NullIoDevice;
	RETURN;
END_IF

FOR i := 0 TO (EcMaster.CfgSlaveCount - 1) DO
	IF IoDevice[i].Name = Name THEN
		GetIoDeviceByName := IoDevice[i];
		RETURN;
	END_IF
END_FOR

GetIoDeviceByName := NullIoDevice;
END_METHOD

{attribute 'monitoring' := 'call'}
PROPERTY LocalAmsNetId : T_AmsNetId
GET
LocalAmsNetId := _LocalAmsNetId;
END_GET
END_PROPERTY

{attribute 'monitoring' := 'call'}
PROPERTY MasterAmsNetId : T_AmsNetId
GET
MasterAmsNetId := _MasterAmsNetId;
END_GET
END_PROPERTY

METHOD RegisterEventProvider
VAR_INPUT
	EventProvider : I_EtherCatDiagnosticEventProvider;
END_VAR
THIS^.EventProvider := EventProvider;
END_METHOD

{attribute 'monitoring' := 'call'}
PROPERTY SlaveCount : UINT
GET
SlaveCount := EcMaster.SlaveCount;
END_GET
END_PROPERTY

METHOD Initialize
VAR_INST
	InitSequenceState : UDINT;
	GetLocalAmsNetId  : FB_GetLocalAmsNetId;
	StartCycles		  : UINT;
END_VAR

VAR
	i : UDINT;
END_VAR
IF NOT _Error AND NOT (F_GetMappingStatus(ADR(EcMaster.AmsNetID), SIZEOF(EcMaster.AmsNetID)) <> EplcMappingStatus.MS_Unmapped) AND NOT Simulated THEN
	_Error := TRUE;
	Trace.LogMessage(Name, 'Init Failed - AmsNetID mapped to Master!');
END_IF

IF NOT _Error AND NOT (F_GetMappingStatus(ADR(EcMaster.DevID), SIZEOF(EcMaster.DevID)) <> EplcMappingStatus.MS_Unmapped) AND NOT Simulated THEN
	_Error := TRUE;
	Trace.LogMessage(Name, 'Init Failed - DevID mapped to Master!');
END_IF

IF NOT _Error AND NOT (F_GetMappingStatus(ADR(EcMaster.DevState), SIZEOF(EcMaster.DevState)) <> EplcMappingStatus.MS_Unmapped) AND NOT Simulated THEN
	_Error := TRUE;
	Trace.LogMessage(Name, 'Init Failed - DevState mapped to Master!');
END_IF

IF NOT _Error AND NOT (F_GetMappingStatus(ADR(EcMaster.ChangeCount), SIZEOF(EcMaster.ChangeCount)) <> EplcMappingStatus.MS_Unmapped) AND NOT Simulated THEN
	_Error := TRUE;
	Trace.LogMessage(Name, 'Init Failed - ChangeCount mapped to Master!');
END_IF

IF NOT _Error AND NOT (F_GetMappingStatus(ADR(EcMaster.SlaveCount), SIZEOF(EcMaster.SlaveCount)) <> EplcMappingStatus.MS_Unmapped) AND NOT Simulated THEN
	_Error := TRUE;
	Trace.LogMessage(Name, 'Init Failed - CfgSlaveCount mapped to Master!');
END_IF

IF NOT _Error AND NOT (F_GetMappingStatus(ADR(EcMaster.CfgSlaveCount), SIZEOF(EcMaster.CfgSlaveCount)) <> EplcMappingStatus.MS_Unmapped) AND NOT Simulated THEN
	_Error := TRUE;
	Trace.LogMessage(Name, 'Init Failed - CfgSlaveCount mapped to Master!');
END_IF

IF _Error THEN
	RETURN;
END_IF

IF Simulated THEN
	FOR i := 0 TO (SYNC_UNITS - 1) DO
		SyncUnit[i].EventProvider := EventProvider;
		SyncUnit[i].Simulated	  := Simulated;
		SyncUnit[i].Initialize();
		IF NOT SyncUnit[i].Initialized THEN
			RETURN;
		END_IF
	END_FOR

	_Initialized := TRUE;
	RETURN;
END_IF

GetLocalAmsNetId(tTimeOut := T#1S);
_MasterAmsNetId := F_CreateAmsNetId(EcMaster.AmsNetID);
GetMasterFrameCount(sNetId := _MasterAmsNetId, tTimeout := T#1S);
GetConfiguredSlaves(sNetId				:= _MasterAmsNetId,
					pArrEcConfSlaveInfo := ADR(ConfiguredSlaveInfo),
					cbBufLen			:= SIZEOF(ConfiguredSlaveInfo),
					tTimeout			:= T#1S);

CASE InitSequenceState OF
	0:
		GetLocalAmsNetId.bExecute := TRUE;
		IF GetLocalAmsNetId.bBusy THEN
			NextMinorStep(InitSequenceState);
		END_IF

	1:
		IF NOT GetLocalAmsNetId.bBusy AND NOT GetLocalAmsNetId.bError THEN
			_LocalAmsNetId := GetLocalAmsNetId.AddrString;
			NextStep(InitSequenceState);
		END_IF

		IF GetLocalAmsNetId.bError THEN
			_ErrorID := GetLocalAmsNetId.nErrId;
			_Error	 := TRUE;
			Trace.LogMessage(Name, 'Init Failed - GetLocalAmsNetId!');
			InitSequenceState := 999;
		END_IF

	10:
		GetConfiguredSlaves.bExecute := TRUE;
		IF GetConfiguredSlaves.bBusy THEN
			NextMinorStep(InitSequenceState);
		END_IF

	11:
		IF NOT GetConfiguredSlaves.bBusy AND NOT GetConfiguredSlaves.bError THEN
			NextStep(InitSequenceState);
		END_IF

		IF GetConfiguredSlaves.bError THEN
			_ErrorId := GetConfiguredSlaves.nErrorId;
			_Error	 := TRUE;
			Trace.LogMessage(Name, 'Init Failed - Configured EtherCat Slaves could not be read - check linking of EtherCat Master FB!');
			InitSequenceState := 999;
		END_IF

	20: // Get Master Frame Count
		GetMasterFrameCount.bExecute := TRUE;
		IF GetMasterFrameCount.bBusy THEN
			NextMinorStep(InitSequenceState);
		END_IF

	21:
		IF NOT GetMasterFrameCount.bBusy AND NOT GetMasterFrameCount.bError THEN
			// Check Frame Count
			IF GetMasterFrameCount.nFrames > FRAMES THEN
				_Error := TRUE;
				Trace.LogMessage(Name, 'Increase of Frame diagnostic array (FRAMES_MAX) and link to FrmXWcState!');
				RETURN;
			END_IF

			// Check Frame Linking
			FOR i := 0 TO (GetMasterFrameCount.nFrames - 1) DO
				IF NOT (F_GetMappingStatus(ADR(FrmXWcState[i]), SIZEOF(FrmXWcState[i])) <> EplcMappingStatus.MS_Unmapped) THEN
					_Error := TRUE;
					Trace.LogMessage(Name, 'Init Failed - FrmXWcState[x] not mapped to Master!');
					RETURN;
				END_IF
			END_FOR

			NextStep(InitSequenceState);
		END_IF

		IF GetMasterFrameCount.bError THEN
			_ErrorId := GetMasterFrameCount.nErrId;
			_Error	 := TRUE;
			Trace.LogMessage(Name, 'Init Failed - Configured EtherCat Frames could not be read!');
			InitSequenceState := 999;
		END_IF

	30:
		FOR i := 0 TO (SYNC_UNITS - 1) DO
			SyncUnit[i].EventProvider := EventProvider;
			SyncUnit[i].Initialize();
			IF NOT SyncUnit[i].Initialized THEN
				RETURN;
			END_IF
		END_FOR

		NextStep(InitSequenceState);

	40:
		StartCycles := StartCycles + 1;
		IF StartCycles = EcStartupCycles THEN
			FOR i := 0 TO (EcMaster.CfgSlaveCount - 1) DO
				IoDevice[i].AmsNetId	  := EcMaster.AmsNetID;
				IoDevice[i].Name		  := ConfiguredSlaveInfo[i].sName;
				IoDevice[i].State		  REF= SlavesState[i];
				IoDevice[i].Configuration REF= ConfiguredSlaveInfo[i];
			END_FOR

			_Initialized := TRUE;
		END_IF

	999: // Fail - Look at trace message in ADS log
END_CASE
END_METHOD

{attribute 'monitoring' := 'call'}
PROPERTY Initialized : BOOL
GET
Initialized := _Initialized;
END_GET
SET
_Initialized := Initialized;
END_SET
END_PROPERTY

METHOD Reset
IF EventProvider <> 0 THEN
	EventProvider.Reset();
END_IF

LastMasterState := 0;
LastChangeCount := 0;
LastSlaveCount	:= 0;
_Error			:= FALSE;
_ErrorId		:= 0;
SlaveSequence	:= 0;
RunSlaveDiag	:= FALSE;
END_METHOD

{attribute 'monitoring' := 'call'}
PROPERTY Busy : BOOL
GET
Busy := _Busy;
END_GET
END_PROPERTY

{attribute 'monitoring' := 'call'}
PROPERTY Error : BOOL
GET
Error := _Error;
END_GET
END_PROPERTY

{attribute 'monitoring' := 'call'}
PROPERTY ErrorId : UDINT
GET
ErrorId := _ErrorId;
END_GET
END_PROPERTY

METHOD CyclicLogic
VAR
	i : UINT;
END_VAR
IF NOT Initialized THEN
	Initialize();
	RETURN;
END_IF

IF Simulated THEN
	_Busy	 := FALSE;
	_Error	 := FALSE;
	_ErrorId := 0;
ELSE
	IF NOT _Busy THEN
		IF (LastChangeCount <> EcMaster.ChangeCount) THEN
			RunSlaveDiag := TRUE;
		ELSIF ((EcMaster.CfgSlaveCount <> EcMaster.SlaveCount) AND (LastSlaveCount <> EcMaster.SlaveCount)) THEN
			RunSlaveDiag := TRUE;
		ELSIF FramesWcStatesOk() <> LastFramesWcStatesOk THEN
			RunSlaveDiag := TRUE;
		END_IF

		IF RunSlaveDiag THEN
			LastChangeCount		 := EcMaster.ChangeCount;
			LastSlaveCount		 := EcMaster.SlaveCount;
			LastFramesWcStatesOk := FramesWcStatesOk();
		END_IF
	END_IF

	GetSlaveTopologyInfo(sNetId	  := _MasterAmsNetId,
						 pAddrBuf := ADR(SlaveTopologyInfo),
						 cbBufLen := SIZEOF(SlaveTopologyInfo),
						 tTimeout := T#5S);

	GetAllSlaveStates(sNetId	:= _MasterAmsNetId,
					  pStateBuf := ADR(SlavesState),
					  cbBufLen	:= SIZEOF(SlavesState),
					  tTimeout	:= T#5S);

	MasterState();
	SlaveState();
	FOR i := 0 TO (SYNC_UNITS - 1) DO
		SyncUnit[i].CyclicLogic();
	END_FOR

	_Busy := SlaveSequence <> 0;
END_IF

FOR i := 0 TO (EcMaster.CfgSlaveCount - 1) DO
	IoDevice[i].CyclicLogic();
END_FOR
END_METHOD

(*FB_Init is always available implicitly and it is used primarily for initialization.
The return value is not evaluated. For a specific influence, you can also declare the
methods explicitly and provide additional code there with the standard initialization
code. You can evaluate the return value.*)
METHOD FB_Init : BOOL
VAR_INPUT
	(* TRUE: the retain variables are initialized (reset warm / reset cold)*)
	bInitRetains : BOOL;

	(* TRUE: the instance will be copied to the copy code afterward (online change)   *)
	bInCopyCode		: BOOL;
	Name			: T_MaxString;
	EcStartupCycles : UINT;
END_VAR
THIS^.EcStartupCycles := EcStartupCycles;
END_METHOD

{attribute 'monitoring' := 'call'}
PROPERTY Simulated : BOOL
GET
Simulated := _Simulated;
END_GET
SET
_Simulated := Simulated;
END_SET
END_PROPERTY

END_FUNCTION_BLOCK

// Components/EtherCat/SyncUnitTask
{attribute 'no_explicit_call' := 'do not call this POU directly'}
FUNCTION_BLOCK FINAL SyncUnitTask EXTENDS CyclicComponent IMPLEMENTS I_SyncUnitTask, I_Initializable, I_TaskResult, I_Simulatable
VAR
	SyncUnitTaskInfo AT %I* : ST_EtherCatSyncUnitTaskInfo;
	_SlaveCount				: UINT;
	_IsHotConnect			: BOOL;
	EcMaster				: I_EtherCatMasterDiagnostic;
	ConfiguredSlaveInfo		: REFERENCE TO ARRAY[0..MAX_EC_SLAVES] OF ST_EcSlaveConfigData;
	SlaveTopologyInfo		: REFERENCE TO ARRAY[0..MAX_EC_SLAVES] OF ST_TopologyDataEx;
	SyncUnitSlaveAddresses	: ARRAY[0..MAX_EC_SLAVES] OF UINT;
	SyncUnitSlaveNames		: ARRAY[0..MAX_EC_SLAVES] OF STRING(31);
END_VAR

VAR
	{attribute 'hide'}
	_Initialized : BOOL;
	{attribute 'hide'}
	_Error : BOOL;
	{attribute 'hide'}
	_Busy : BOOL;
	{attribute 'hide'}
	_ErrorId : UDINT;
	{attribute 'hide'}
	_Simulated : BOOL;
END_VAR

VAR
	SyncUnitState			  : UDINT := READ_SLAVES;
	i						  : UINT;
	j						  : UINT;
	_EventProvider			  : I_EtherCatDiagnosticEventProvider;
	EcGetAllSyncUnitSlaveAddr : FB_EcGetAllSyncUnitSlaveAddr;
END_VAR

VAR CONSTANT
	ERROR_READ_SLAVE_NAMES	   : UDINT := 1;
	ERROR_REGISTER_SYNC_UNIT   : UDINT := 2;
	ERROR_VALID_DATA_SYNC_UNIT : UDINT := 3;
	STRING_LEN				   : INT   := 80;
	SYNC_UNIT_ALARM_MAX		   : UINT  := 3;

	//
	READ_SLAVES			  : UDINT := 0;
	READ_SLAVES_DONE	  : UDINT := 1;
	SYNC_UNIT_OK		  : UDINT := 2;
	POPULATE_SLAVE_NAMES  : UDINT := 3;
	WORKING_COUNTER_ERROR : UDINT := 4;
	READ_ERROR			  : UDINT := 5;
END_VAR

METHOD Initialize
VAR_INPUT
END_VAR
IF NOT _Error AND NOT (F_GetMappingStatus(ADR(SyncUnitTaskInfo.ObjectId), SIZEOF(SyncUnitTaskInfo.ObjectId)) <> EplcMappingStatus.MS_Unmapped) AND NOT Simulated THEN
	_Error := TRUE;
	Trace.LogMessage(Name, 'Init Failed - SyncUnitTaskInfo.ObjectId mapped to SyncUnit Diagnostic!');
END_IF

IF NOT _Error AND NOT (F_GetMappingStatus(ADR(SyncUnitTaskInfo.SlaveCount), SIZEOF(SyncUnitTaskInfo.SlaveCount)) <> EplcMappingStatus.MS_Unmapped) AND NOT Simulated THEN
	_Error := TRUE;
	Trace.LogMessage(Name, 'Init Failed - SyncUnitTaskInfo.SlaveCount mapped to SyncUnit Diagnostic!');
END_IF

IF NOT _Error AND NOT (F_GetMappingStatus(ADR(SyncUnitTaskInfo.State), SIZEOF(SyncUnitTaskInfo.State)) <> EplcMappingStatus.MS_Unmapped) AND NOT Simulated THEN
	_Error := TRUE;
	Trace.LogMessage(Name, 'Init Failed - SyncUnitTaskInfo.State mapped to SyncUnit Diagnostic!');
END_IF

IF NOT _Error AND NOT (F_GetMappingStatus(ADR(SyncUnitTaskInfo.WcState), SIZEOF(SyncUnitTaskInfo.WcState)) <> EplcMappingStatus.MS_Unmapped) AND NOT Simulated THEN
	_Error := TRUE;
	Trace.LogMessage(Name, 'Init Failed - SyncUnitTaskInfo.WcState mapped to SyncUnit Diagnostic!');
END_IF

IF _Error THEN
	RETURN;
END_IF

IF Simulated THEN
	_Initialized := TRUE;
	RETURN;
END_IF

F_EcGetSyncUnitName(SyncUnitTaskInfo.ObjectId, sSyncUnitName => _Name);
_Initialized := TRUE;
END_METHOD

{attribute 'monitoring' := 'call'}
PROPERTY Initialized : BOOL
GET
Initialized := _Initialized;
END_GET
SET
_Initialized := Initialized;
END_SET
END_PROPERTY

{attribute 'monitoring' := 'call'}
PROPERTY IoDataValid : BOOL
GET
IoDataValid := NOT SyncUnitTaskInfo.WcState;
END_GET
END_PROPERTY

{attribute 'monitoring' := 'call'}
PROPERTY IsHotConnect : BOOL
GET
IsHotConnect := _IsHotConnect;
END_GET
END_PROPERTY

METHOD IsTerminalPartOfSyncUnit : BOOL
VAR_INPUT
	Addr : UINT;
END_VAR
FOR i := 0 TO (_SlaveCount - 1) DO
	IF SyncUnitSlaveAddresses[i] = Addr THEN
		IsTerminalPartOfSyncUnit := TRUE;
		EXIT;
	END_IF
END_FOR
END_METHOD

{attribute 'monitoring' := 'call'}
PROPERTY PUBLIC SlaveCount : UINT
GET
SlaveCount := _SlaveCount;
END_GET
END_PROPERTY

{attribute 'monitoring' := 'call'}
PROPERTY Busy : BOOL
GET
Busy := _Busy;
END_GET
END_PROPERTY

{attribute 'monitoring' := 'call'}
PROPERTY Error : BOOL
GET
Error := _Error;
END_GET
END_PROPERTY

{attribute 'monitoring' := 'call'}
PROPERTY ErrorId : UDINT
GET
ErrorId := _ErrorId;
END_GET
END_PROPERTY

METHOD PUBLIC CyclicLogic
VAR_INST
	TempSlaveMessage  : STRING;
	SlaveMessagePartA : STRING;
	SlaveMessagePartB : STRING;
END_VAR
IF NOT Initialized THEN
	Initialize();
	RETURN;
END_IF

IF Simulated THEN
	RETURN;
END_IF

EcGetAllSyncUnitSlaveAddr(sNetId	:= '',
						  nObjectId := SyncUnitTaskInfo.ObjectId,
						  pAddrBuf	:= ADR(SyncUnitSlaveAddresses),
						  cbBufLen	:= (SIZEOF(UINT) * MAX_EC_SLAVES),
						  tTimeout	:= T#5S,
						  nSlaves	=> _SlaveCount);

EcGetAllSyncUnitSlaveAddr.bExecute := FALSE;
CASE SyncUnitState OF
	READ_SLAVES:
		EcGetAllSyncUnitSlaveAddr.bExecute := TRUE;
		SyncUnitState					   := READ_SLAVES_DONE;

	READ_SLAVES_DONE:
		IF NOT EcGetAllSyncUnitSlaveAddr.bBusy AND NOT EcGetAllSyncUnitSlaveAddr.bError AND (_SlaveCount > 0) THEN
			SyncUnitState := POPULATE_SLAVE_NAMES;
		END_IF

		IF (EcGetAllSyncUnitSlaveAddr.bError OR (_SlaveCount = 0)) AND NOT EcGetAllSyncUnitSlaveAddr.bBusy THEN
			SyncUnitState := READ_ERROR;
		END_IF

	POPULATE_SLAVE_NAMES:
		FOR i := 0 TO (_SlaveCount - 1) DO
			FOR j := 0 TO (EcMaster.ConfiguredSlaveCount - 1) DO
				IF SyncUnitSlaveAddresses[i] <> 0 THEN
					IF SyncUnitSlaveAddresses[i] = ConfiguredSlaveInfo[j].nAddr THEN
						_IsHotConnect		  := SlaveTopologyInfo[j].nStatusBits.4 OR SlaveTopologyInfo[j].nStatusBits.5;
						SyncUnitSlaveNames[i] := ConfiguredSlaveInfo[j].sName;
					END_IF
				END_IF
			END_FOR
		END_FOR

		TempSlaveMessage  := '';
		SlaveMessagePartA := '';
		SlaveMessagePartB := '';
		FOR j := 0 TO (_SlaveCount - 1) DO
			IF LEN(SyncUnitSlaveNames[j]) > 0 THEN
				TempSlaveMessage := CONCAT(SyncUnitSlaveNames[j], ', ');
				IF (LEN(TempSlaveMessage) + LEN(SlaveMessagePartA)) <= STRING_LEN THEN
					SlaveMessagePartA := CONCAT(SlaveMessagePartA, TempSlaveMessage);
				ELSIF (LEN(TempSlaveMessage) + LEN(SlaveMessagePartB)) <= STRING_LEN THEN
					SlaveMessagePartB := CONCAT(SlaveMessagePartB, TempSlaveMessage);
				END_IF
			END_IF
		END_FOR

		SyncUnitState := SYNC_UNIT_OK;

	SYNC_UNIT_OK:
		IF SyncUnitTaskInfo.WcState THEN
			SyncUnitState := WORKING_COUNTER_ERROR;
			_Busy		  := TRUE;
		ELSE
			_Error	 := FALSE;
			_ErrorID := 0;
			_Busy	 := FALSE;
		END_IF

	WORKING_COUNTER_ERROR:
		_Busy	 := FALSE;
		_Error	 := TRUE;
		_ErrorID := ERROR_VALID_DATA_SYNC_UNIT;
		IF _EventProvider <> 0 THEN
			IF _IsHotConnect THEN
				_EventProvider.RaiseSyncUnitEvent(E_SyncUnit.SyncUnitWarning,
												  _Name,
												  SlaveMessagePartA,
												  SlaveMessagePartB);
			ELSIF NOT _IsHotConnect THEN
				_EventProvider.RaiseSyncUnitEvent(E_SyncUnit.SyncUnitError,
												  _Name,
												  SlaveMessagePartA,
												  SlaveMessagePartB);
			END_IF
		END_IF

		IF NOT SyncUnitTaskInfo.WcState THEN
			IF _EventProvider <> 0 THEN
				_EventProvider.Reset();
			END_IF

			SyncUnitState := READ_SLAVES;
		END_IF

	READ_ERROR:
		Trace.LogMessage(Name, CONCAT('Sync Unit Slave Names could not be read! Error ID: ', TO_STRING(EcGetAllSyncUnitSlaveAddr.nErrId)));
		_Error		  := TRUE;
		_ErrorID	  := ERROR_READ_SLAVE_NAMES;
		SyncUnitState := READ_SLAVES;
END_CASE
END_METHOD

PROPERTY EventProvider : I_EtherCatDiagnosticEventProvider
SET
_EventProvider := EventProvider;
END_SET
END_PROPERTY

(*FB_Init is always available implicitly and it is used primarily for initialization.
The return value is not evaluated. For a specific influence, you can also declare the
methods explicitly and provide additional code there with the standard initialization
code. You can evaluate the return value.*)
METHOD FB_Init : BOOL
VAR_INPUT
	(* TRUE: the retain variables are initialized (reset warm / reset cold)*)
	bInitRetains : BOOL;

	(* TRUE: the instance will be copied to the copy code afterward (online change)   *)
	bInCopyCode			: BOOL;
	Name				: T_MaxString;
	EcMaster			: I_EtherCatMasterDiagnostic;
	ConfiguredSlaveInfo : REFERENCE TO ARRAY[0..MAX_EC_SLAVES] OF ST_EcSlaveConfigData;
	SlaveTopologyInfo	: REFERENCE TO ARRAY[0..MAX_EC_SLAVES] OF ST_TopologyDataEx;
END_VAR
THIS^.EcMaster			  := EcMaster;
THIS^.ConfiguredSlaveInfo REF= ConfiguredSlaveInfo;
THIS^.SlaveTopologyInfo	  REF= SlaveTopologyInfo;
END_METHOD

{attribute 'monitoring' := 'call'}
PROPERTY Simulated : BOOL
GET
Simulated := _Simulated;
END_GET
SET
_Simulated := Simulated;
END_SET
END_PROPERTY

END_FUNCTION_BLOCK

// Statemachine/Generic/NextStep
FUNCTION NextStep : UDINT
VAR_IN_OUT
	StateVar : UDINT;
END_VAR

NextStep := StateVar := ((StateVar / 10) * 10) + 10;

END_FUNCTION

// Statemachine/Generic/NextMinorStep
FUNCTION NextMinorStep : UDINT
VAR_IN_OUT
	StateVar : UDINT;
END_VAR

NextMinorStep := StateVar := StateVar + 1;

END_FUNCTION

// Components/EtherCat/EtherCatMaster_TcEvents
FUNCTION_BLOCK EtherCatMaster_TcEvents EXTENDS Component IMPLEMENTS I_EtherCatDiagnosticEventProvider
VAR
	EtherCatMasterDiagnostic : I_EtherCatMasterDiagnostic;
	SyncUnitEvents			 : TcEventClass('Sync Unit Events');
	EtherCatMasterEvents	 : TcEventClass('EtherCAT Master Events');
END_VAR

METHOD GetHighestActiveEventReaction : DINT
GetHighestActiveEventReaction := MAX(EtherCatMasterEvents.GetHighestActiveEventReaction(), SyncUnitEvents.GetHighestActiveEventReaction());
END_METHOD

METHOD GetHighestActiveEventSeverity : TcEventSeverity
GetHighestActiveEventSeverity := MAX(SyncUnitEvents.GetHighestActiveEventSeverity(), EtherCatMasterEvents.GetHighestActiveEventSeverity());
END_METHOD

METHOD RaiseEtherCatDiagnosticEvent
VAR_INPUT
	EventId	  : UDINT;
	Argument1 : STRING := '';
	Argument2 : STRING := '';
	Argument3 : STRING := '';
END_VAR
IF Argument3 <> '' THEN
	EtherCatMasterEvents.Arguments(EventId).Clear().AddString(Argument1).AddString(Argument2).AddString(Argument3);
ELSIF Argument2 <> '' THEN
	EtherCatMasterEvents.Arguments(EventId).Clear().AddString(Argument1).AddString(Argument2);
ELSIF Argument1 <> '' THEN
	EtherCatMasterEvents.Arguments(EventId).Clear().AddString(Argument1);
ELSE
	EtherCatMasterEvents.Arguments(EventId).Clear();
END_IF

EtherCatMasterEvents.RaiseEvent(EventId);
END_METHOD

METHOD RaiseSyncUnitEvent
VAR_INPUT
	EventId	  : UDINT;
	Argument1 : STRING := '';
	Argument2 : STRING := '';
	Argument3 : STRING := '';
END_VAR
IF Argument3 <> '' THEN
	SyncUnitEvents.Arguments(EventId).Clear().AddString(Argument1).AddString(Argument2).AddString(Argument3);
ELSIF Argument2 <> '' THEN
	SyncUnitEvents.Arguments(EventId).Clear().AddString(Argument1).AddString(Argument2);
ELSIF Argument1 <> '' THEN
	SyncUnitEvents.Arguments(EventId).Clear().AddString(Argument1);
ELSE
	SyncUnitEvents.Arguments(EventId).Clear();
END_IF

SyncUnitEvents.RaiseEvent(EventId);
END_METHOD

METHOD Reset
SyncUnitEvents.Reset();
EtherCatMasterEvents.Reset();
END_METHOD

METHOD SetEventReactions
VAR_INPUT
	Verbose	 : DINT := 0;
	Info	 : DINT := 1;
	Warning	 : DINT := 2;
	Error	 : DINT := 3;
	Critical : DINT := 4;
END_VAR
SyncUnitEvents.SetEventReactions(Verbose,
								 Info,
								 Warning,
								 Error,
								 Critical);

EtherCatMasterEvents.SetEventReactions(Verbose,
									   Info,
									   Warning,
									   Error,
									   Critical);
END_METHOD

(*FB_Init is always available implicitly and it is used primarily for initialization.
The return value is not evaluated. For a specific influence, you can also declare the
methods explicitly and provide additional code there with the standard initialization
code. You can evaluate the return value.*)
METHOD FB_Init : BOOL
VAR_INPUT
	(* TRUE: the retain variables are initialized (reset warm / reset cold)*)
	bInitRetains : BOOL;

	(* TRUE: the instance will be copied to the copy code afterward (online change)   *)
	bInCopyCode				 : BOOL;
	Name					 : T_MaxString;
	EtherCatMasterDiagnostic : I_EtherCatMasterDiagnostic;
END_VAR
THIS^.EtherCatMasterDiagnostic := EtherCatMasterDiagnostic;
THIS^.EtherCatMasterDiagnostic.RegisterEventProvider(THIS^);
SyncUnitEvents.GenerateTcEvents(EtherCatMasterDiagnostic.Name, ADR(TC_Events.SyncUnit), SIZEOF(ST_SyncUnit));
EtherCatMasterEvents.GenerateTcEvents(EtherCatMasterDiagnostic.Name, ADR(TC_Events.EtherCatMaster), SIZEOF(ST_EtherCatMaster));
END_METHOD

END_FUNCTION_BLOCK

// Components/Recipe/Interface/I_RecipeManagment
INTERFACE I_RecipeManagment EXTENDS I_Component

{attribute 'monitoring' := 'call'}
PROPERTY AutoLoadChangesToActive : BOOL
SET
END_SET
END_PROPERTY

{attribute 'monitoring' := 'call'}
PROPERTY ChangesPending : BOOL
GET
END_GET
END_PROPERTY

METHOD LoadChangesToActive
VAR_INPUT
END_VAR
END_METHOD

END_INTERFACE

// Components/Recipe/RecipeManagment
FUNCTION_BLOCK RecipeManagment EXTENDS CyclicComponent IMPLEMENTS I_RecipeManagment
VAR
	nRecipe					 : UDINT;
	pActiveRecipeData		 : PVOID;
	pUpdateRecipeData		 : PVOID;
	_ChangesPending			 : BOOL;
	_AutoLoadChangesToActive : BOOL;
END_VAR

METHOD CyclicLogic
IF nRecipe = 0 THEN
	RETURN;
END_IF

IF pActiveRecipeData = 0 THEN
	RETURN;
END_IF

IF pUpdateRecipeData = 0 THEN
	RETURN;
END_IF

CompareData();
END_METHOD

METHOD CompareData
VAR_INPUT
END_VAR
IF MEMCMP(pActiveRecipeData, pUpdateRecipeData, nRecipe) = 0 THEN
	_ChangesPending := FALSE;
ELSE
	IF _AutoLoadChangesToActive THEN
		LoadChangesToActive();
	ELSE
		_ChangesPending := TRUE;
	END_IF
END_IF
END_METHOD

{attribute 'monitoring' := 'call'}
PROPERTY AutoLoadChangesToActive : BOOL
SET
_AutoLoadChangesToActive := AutoLoadChangesToActive;
END_SET
END_PROPERTY

{attribute 'monitoring' := 'call'}
PROPERTY ChangesPending : BOOL
GET
ChangesPending := _ChangesPending;
END_GET
END_PROPERTY

METHOD LoadChangesToActive
VAR_INPUT
END_VAR
MEMCPY(pActiveRecipeData, pUpdateRecipeData, nRecipe);
CompareData();
END_METHOD

(*FB_Init is always available implicitly and it is used primarily for initialization.
The return value is not evaluated. For a specific influence, you can also declare the
methods explicitly and provide additional code there with the standard initialization
code. You can evaluate the return value.*)
METHOD FB_Init : BOOL
VAR_INPUT
	(* TRUE: the retain variables are initialized (reset warm / reset cold)*)
	bInitRetains : BOOL;

	(* TRUE: the instance will be copied to the copy code afterward (online change)   *)
	bInCopyCode		  : BOOL;
	Name			  : T_MaxString;
	nRecipe			  : UDINT;
	pActiveRecipeData : PVOID;
	pUpdateRecipeData : PVOID;
END_VAR
THIS^.nRecipe			:= nRecipe;
THIS^.pActiveRecipeData := pActiveRecipeData;
THIS^.pUpdateRecipeData := pUpdateRecipeData;
END_METHOD

END_FUNCTION_BLOCK

// Components/Safety/Interface/I_InSafetyGroup
INTERFACE I_InSafetyGroup EXTENDS I_Base

PROPERTY SafetyGroup : I_TaskResult
SET
END_SET
END_PROPERTY

END_INTERFACE

// Components/Safety/Interface/I_SafetyBase
INTERFACE I_SafetyBase EXTENDS I_Component, I_Resettable, I_SafetySimulation, I_TaskResult

{attribute 'monitoring' := 'call'}
PROPERTY OK : BOOL
GET
END_GET
END_PROPERTY

PROPERTY ResetFunction : I_SafetyReset
SET
END_SET
END_PROPERTY

END_INTERFACE

// Components/Safety/Interface/I_SafetySimulation
INTERFACE I_SafetySimulation EXTENDS I_Simulatable

METHOD SimulateSafetyDiag
VAR_INPUT
	SimulationValueDiag : UINT;
END_VAR
END_METHOD

METHOD SimulateSafetyState
VAR_INPUT
	SimulationValueState : USINT;
END_VAR
END_METHOD

END_INTERFACE

// Components/Safety/Interface/I_SafetyReset
INTERFACE I_SafetyReset EXTENDS I_Cyclic, I_TaskResult

METHOD Execute
VAR_INPUT
END_VAR
END_METHOD

PROPERTY PulseDuration : TIME
SET
END_SET
END_PROPERTY

END_INTERFACE

// Components/Safety/Interface/I_SafetyModule
INTERFACE I_SafetyModule EXTENDS I_SafetySimulation, I_TaskResult, I_Resettable, I_Module

METHOD AddSafetyComponent
VAR_INPUT
	Component : I_SafetyBase;
END_VAR
END_METHOD

{attribute 'monitoring' := 'call'}
PROPERTY OK : BOOL
GET
END_GET
END_PROPERTY

PROPERTY SafetyPlcCoE : I_CoeDevice
GET
END_GET
END_PROPERTY

END_INTERFACE

// Components/Safety/Reset Function/SafetyResetPulse
FUNCTION_BLOCK SafetyResetPulse EXTENDS CyclicComponent IMPLEMENTS I_SafetyReset
VAR
	Reset AT %Q*   : BOOL;
	TpErrorAck	   : TP;
	TofErrorAck	   : TOF;
	_PulseDuration : TIME := T#100MS;
	_Error		   : BOOL;
	_Busy		   : BOOL;
END_VAR

METHOD CyclicLogic
TpErrorAck(PT := _PulseDuration, Q => Reset);
IF TpErrorAck.Q THEN
	TpErrorAck.IN := FALSE;
END_IF

TofErrorAck(In := TpErrorAck.Q, PT := _PulseDuration);
_Error := FALSE;
_Busy  := TofErrorAck.Q;
END_METHOD

{attribute 'monitoring' := 'call'}
PROPERTY Busy : BOOL
GET
Busy := _Busy;
END_GET
END_PROPERTY

{attribute 'monitoring' := 'call'}
PROPERTY Error : BOOL
GET
Error := _Error;
END_GET
END_PROPERTY

{attribute 'monitoring' := 'call'}
PROPERTY ErrorId : UDINT
GET
END_GET
END_PROPERTY

METHOD Execute
IF TpErrorAck.Q THEN
	RETURN;
END_IF

TpErrorAck.IN := TRUE;
END_METHOD

PROPERTY PulseDuration : TIME
SET
_PulseDuration := PulseDuration;
END_SET
END_PROPERTY

END_FUNCTION_BLOCK

// Components/Safety/Visitor/SafetyOkVisitor
FUNCTION_BLOCK SafetyOkVisitor IMPLEMENTS I_ComponentVisitor
VAR
	{attribute 'hide'}
	_OK				: BOOL;
	SafetyComponent : I_SafetyBase;
	ErrorComponent	: I_Component;
END_VAR

METHOD Check
VAR_INPUT
	Components : I_ComponentCollection;
END_VAR
_OK := TRUE;
Components.Accept(THIS^);
END_METHOD

{attribute 'monitoring' := 'call'}
PROPERTY OK : BOOL
GET
OK := _OK;
END_GET
END_PROPERTY

METHOD VisitComponent
VAR_INPUT
	Component : I_Component;
END_VAR
IF __QUERYINTERFACE(Component, SafetyComponent) THEN
	IF NOT SafetyComponent.OK THEN
		ErrorComponent := Component;
		_OK			   := FALSE;
	END_IF
END_IF
END_METHOD

END_FUNCTION_BLOCK

// Components/Safety/Visitor/SetSafetySimulationVisitor
FUNCTION_BLOCK SetSafetySimulationVisitor IMPLEMENTS I_ComponentVisitor
VAR
	SafetyComponent : I_SafetyBase;
	InfoData		: ST_SafetyStateDiag;
	_Simulated		: BOOL;
END_VAR

PROPERTY Diag : UINT
SET
InfoData.Diag := Diag;
END_SET
END_PROPERTY

PROPERTY Simulated : BOOL
GET
Simulated := _Simulated;
END_GET
SET
_Simulated := Simulated;
END_SET
END_PROPERTY

PROPERTY State : USINT
SET
InfoData.State := State;
END_SET
END_PROPERTY

METHOD VisitComponent
VAR_INPUT
	Component : I_Component;
END_VAR
IF __QUERYINTERFACE(Component, SafetyComponent) THEN
	SafetyComponent.Simulated := _Simulated;
	SafetyComponent.SimulateSafetyDiag(InfoData.Diag);
	SafetyComponent.SimulateSafetyState(InfoData.State);
END_IF
END_METHOD

END_FUNCTION_BLOCK

// Components/Safety/SafetyAndOrFB
FUNCTION_BLOCK SafetyAndOrFB EXTENDS SafetyBase
VAR
END_VAR

METHOD CyclicLogic
VAR_INST
END_VAR
SUPER^.CyclicLogic();
_OK := SUPER^.InfoData.State = E_SafetyOrAnd_State.Run;
END_METHOD

END_FUNCTION_BLOCK

// Components/Safety/SafetyBase
FUNCTION_BLOCK SafetyBase EXTENDS CyclicComponent IMPLEMENTS I_SafetyBase
VAR
	InfoData AT %I* : ST_SafetyStateDiag;
	{attribute 'hide'}
	_Simulated : BOOL;
	{attribute 'hide'}
	_OK : BOOL;
	{attribute 'hide'}
	_Error : BOOL;
	{attribute 'hide'}
	_Busy : BOOL;
	{attribute 'hide'}
	_ErrorId	   : UDINT;
	_ResetFunction : I_SafetyReset;
END_VAR

METHOD CyclicLogic
VAR_INST
	LinkError : BOOL;
END_VAR
IF NOT LinkError AND NOT Simulated AND (F_GetMappingStatus(ADR(InfoData), SIZEOF(InfoData)) = EplcMappingStatus.MS_Unmapped) THEN
	LinkError := TRUE;
	Trace.LogMessage(Name, 'Not mapped to Safety, no diagnostics available!');
END_IF

IF _ResetFunction <> 0 THEN
	_ResetFunction.CyclicLogic();
END_IF
END_METHOD

{attribute 'monitoring' := 'call'}
PROPERTY OK : BOOL
GET
OK := _OK;
END_GET
END_PROPERTY

METHOD Reset
IF _ResetFunction <> 0 THEN
	_ResetFunction.Execute();
END_IF
END_METHOD

PROPERTY ResetFunction : I_SafetyReset
SET
_ResetFunction := ResetFunction;
END_SET
END_PROPERTY

{attribute 'monitoring' := 'call'}
PROPERTY Simulated : BOOL
GET
Simulated := _Simulated;
END_GET
SET
_Simulated := Simulated;
END_SET
END_PROPERTY

METHOD SimulateSafetyDiag
VAR_INPUT
	SimulationValueDiag : UINT;
END_VAR
Infodata.Diag := SimulationValueDiag;
END_METHOD

METHOD SimulateSafetyState
VAR_INPUT
	SimulationValueState : USINT;
END_VAR
Infodata.State := SimulationValueState;
END_METHOD

{attribute 'monitoring' := 'call'}
PROPERTY Busy : BOOL
GET
Busy := _Busy;
END_GET
END_PROPERTY

{attribute 'monitoring' := 'call'}
PROPERTY Error : BOOL
GET
Error := _Error;
END_GET
END_PROPERTY

{attribute 'monitoring' := 'call'}
PROPERTY ErrorId : UDINT
GET
ErrorId := _ErrorId;
END_GET
END_PROPERTY

END_FUNCTION_BLOCK

// Components/Safety/SafetyConnectionFB_TcEvents
FUNCTION_BLOCK SafetyConnectionFB_TcEvents EXTENDS SafetyBase IMPLEMENTS I_EventReactionTcEvents
VAR
	Events : TcEventClass('FSoE Connection Events');
END_VAR

METHOD CyclicLogic
VAR_INST
	DiagWord	: WORD;
	BitMaskDiag : WORD := 16#000F;
END_VAR
SUPER^.CyclicLogic();
_OK	   := SUPER^.InfoData.State = E_SafetyConnection_State.Data;
_Error := GetHighestActiveEventReaction() >= TcEventSeverity.Error;
IF _ResetFunction <> 0 AND_THEN _ResetFunction.Busy THEN
	RETURN;
END_IF

BitMaskDiag := 16#000F;
DiagWord	:= TO_WORD(SUPER^.InfoData.Diag) AND BitMaskDiag;
IF (DiagWord = 1) THEN
	Events.RaiseEvent(E_SafetyConnection.InvalidCommand);
END_IF

IF (DiagWord = 2) THEN
	Events.RaiseEvent(E_SafetyConnection.UnknownCommand);
END_IF

IF (DiagWord = 3) THEN
	Events.RaiseEvent(E_SafetyConnection.InvalidConID);
END_IF

IF (DiagWord = 4) THEN
	Events.RaiseEvent(E_SafetyConnection.InvalidCrc);
END_IF

IF (DiagWord = 5) THEN
	Events.RaiseEvent(E_SafetyConnection.WatchdogExpired);
END_IF

IF (DiagWord = 6) THEN
	Events.RaiseEvent(E_SafetyConnection.InvalidFSOEAddr);
END_IF

IF (DiagWord = 7) THEN
	Events.RaiseEvent(E_SafetyConnection.InvalidData);
END_IF

IF (DiagWord = 8) THEN
	Events.RaiseEvent(E_SafetyConnection.InvalidComParameterLen);
END_IF

IF (DiagWord = 9) THEN
	Events.RaiseEvent(E_SafetyConnection.InavlidComParameter);
END_IF

IF (DiagWord = 10) THEN
	Events.RaiseEvent(E_SafetyConnection.InvalidUserParameterLen);
END_IF

IF (DiagWord = 11) THEN
	Events.RaiseEvent(E_SafetyConnection.InvalidUserParameter);
END_IF

IF (DiagWord = 12) THEN
	Events.RaiseEvent(E_SafetyConnection.FSoEMasterReset);
END_IF

IF (DiagWord = 13) THEN
	Events.RaiseEvent(E_SafetyConnection.ModuleErrorOnSlave);
END_IF

IF (DiagWord = 14) THEN
	Events.RaiseEvent(E_SafetyConnection.ModuleError);
END_IF

IF (DiagWord = 15) THEN
	Events.RaiseEvent(E_SafetyConnection.SlaveNotStarted);
END_IF

BitMaskDiag := 16#0010;
DiagWord	:= TO_WORD(SUPER^.InfoData.Diag) AND BitMaskDiag;
IF DiagWord.4 THEN
	Events.RaiseEvent(E_SafetyConnection.FsoESlaveError);
END_IF

BitMaskDiag := 16#0020;
DiagWord	:= TO_WORD(SUPER^.InfoData.Diag) AND BitMaskDiag;
IF DiagWord.5 THEN
	Events.RaiseEvent(E_SafetyConnection.FsoESlaveFailSafeValue);
END_IF

BitMaskDiag := 16#0040;
DiagWord	:= TO_WORD(SUPER^.InfoData.Diag) AND BitMaskDiag;
IF DiagWord.6 THEN
	Events.RaiseEvent(E_SafetyConnection.Startup);
END_IF

BitMaskDiag := 16#0080;
DiagWord	:= TO_WORD(SUPER^.InfoData.Diag) AND BitMaskDiag;
IF DiagWord.7 THEN
	Events.RaiseEvent(E_SafetyConnection.FsoEMasterSafeValue);
END_IF
END_METHOD

METHOD GetHighestActiveEventReaction : DINT
GetHighestActiveEventReaction := Events.GetHighestActiveEventReaction();
END_METHOD

METHOD GetHighestActiveEventSeverity : TcEventSeverity
GetHighestActiveEventSeverity := Events.GetHighestActiveEventSeverity();
END_METHOD

METHOD Reset
SUPER^.Reset();
Events.Reset();
END_METHOD

METHOD SetEventReactions
VAR_INPUT
	Verbose	 : DINT := 0;
	Info	 : DINT := 1;
	Warning	 : DINT := 2;
	Error	 : DINT := 3;
	Critical : DINT := 4;
END_VAR
Events.SetEventReactions(Verbose,
						 Info,
						 Warning,
						 Error,
						 Critical);
END_METHOD

(*FB_Init is always available implicitly and it is used primarily for initialization.
The return value is not evaluated. For a specific influence, you can also declare the
methods explicitly and provide additional code there with the standard initialization
code. You can evaluate the return value.*)
METHOD FB_Init : BOOL
VAR_INPUT
	(* TRUE: the retain variables are initialized (reset warm / reset cold)*)
	bInitRetains : BOOL;

	(* TRUE: the instance will be copied to the copy code afterward (online change)   *)
	bInCopyCode : BOOL;
	Name		: T_MaxString;
END_VAR
Events.GenerateTcEvents(Name, ADR(TC_events.SafetyConnection), SIZEOF(ST_SafetyConnection));
END_METHOD

END_FUNCTION_BLOCK

// Components/Safety/SafetyEdmFB_TcEvents
FUNCTION_BLOCK SafetyEdmFB_TcEvents EXTENDS SafetyBase IMPLEMENTS I_EventReactionTcEvents, I_InSafetyGroup
VAR
	Events		 : TcEventClass('Safety EDM Events');
	_SafetyGroup : I_TaskResult;
END_VAR

METHOD CyclicLogic
SUPER^.CyclicLogic();
_OK	   := SUPER^.InfoData.State <> E_SafetyEdm_State.Error;
_Error := GetHighestActiveEventReaction() >= TcEventSeverity.Error;
IF _SafetyGroup <> 0 THEN
	IF _SafetyGroup.Error THEN
		Events.Reset();
		RETURN;
	END_IF
END_IF

IF _ResetFunction <> 0 AND_THEN _ResetFunction.Busy THEN
	RETURN;
END_IF

IF SUPER^.InfoData.Diag.0 THEN
	Events.RaiseEvent(E_SafetyEdm.SwitchOffTime);
END_IF

IF SUPER^.InfoData.Diag.1 THEN
	Events.RaiseEvent(E_SafetyEdm.SwitchOnTime);
END_IF
END_METHOD

METHOD GetHighestActiveEventReaction : DINT
GetHighestActiveEventReaction := Events.GetHighestActiveEventReaction();
END_METHOD

METHOD GetHighestActiveEventSeverity : TcEventSeverity
GetHighestActiveEventSeverity := Events.GetHighestActiveEventSeverity();
END_METHOD

METHOD Reset
SUPER^.Reset();
Events.Reset();
END_METHOD

METHOD SetEventReactions
VAR_INPUT
	Verbose	 : DINT := 0;
	Info	 : DINT := 1;
	Warning	 : DINT := 2;
	Error	 : DINT := 3;
	Critical : DINT := 4;
END_VAR
Events.SetEventReactions(Verbose,
						 Info,
						 Warning,
						 Error,
						 Critical);
END_METHOD

(*FB_Init is always available implicitly and it is used primarily for initialization.
The return value is not evaluated. For a specific influence, you can also declare the
methods explicitly and provide additional code there with the standard initialization
code. You can evaluate the return value.*)
METHOD FB_Init : BOOL
VAR_INPUT
	(* TRUE: the retain variables are initialized (reset warm / reset cold)*)
	bInitRetains : BOOL;

	(* TRUE: the instance will be copied to the copy code afterward (online change)   *)
	bInCopyCode : BOOL;
	Name		: T_MaxString;
END_VAR
Events.GenerateTcEvents(Name, ADR(TC_events.SafetyEdm), SIZEOF(ST_SafetyEdm));
END_METHOD

PROPERTY SafetyGroup : I_TaskResult
SET
_SafetyGroup := SafetyGroup;
END_SET
END_PROPERTY

END_FUNCTION_BLOCK

// Components/Safety/SafetyEstopFB_TcEvents
FUNCTION_BLOCK SafetyEstopFB_TcEvents EXTENDS SafetyBase IMPLEMENTS I_EventReactionTcEvents, I_InSafetyGroup
VAR
	{attribute 'hide'}
	_ActiveName	 : STRING := 'pressed!';
	Events		 : TcEventClass('Safety E-Stop Events');
	_SafetyGroup : I_TaskResult;
END_VAR

METHOD CyclicLogic
SUPER^.CyclicLogic();
_OK	   := SUPER^.InfoData.State = E_SafetyEStop_State.Run;
_Error := GetHighestActiveEventReaction() >= TcEventSeverity.Error;
IF _SafetyGroup <> 0 THEN
	IF _SafetyGroup.Error THEN
		Events.Reset();
		RETURN;
	END_IF
END_IF

IF _ResetFunction <> 0 AND_THEN _ResetFunction.Busy THEN
	RETURN;
END_IF

IF NOT SUPER^.OK THEN
	Events.Arguments(E_SafetyEstop.Active).Clear().AddString(_ActiveName);
	Events.RaiseEvent(E_SafetyEstop.Active);
END_IF

IF SUPER^.InfoData.Diag.0 THEN
	Events.RaiseEvent(E_SafetyEstop.Disc1);
END_IF

IF SUPER^.InfoData.Diag.1 THEN
	Events.RaiseEvent(E_SafetyEstop.Disc2);
END_IF

IF SUPER^.InfoData.Diag.2 THEN
	Events.RaiseEvent(E_SafetyEstop.Disc3);
END_IF

IF SUPER^.InfoData.Diag.3 THEN
	Events.RaiseEvent(E_SafetyEstop.Disc4);
END_IF

IF SUPER^.InfoData.Diag.4 THEN
	Events.RaiseEvent(E_SafetyEstop.EDM1);
END_IF

IF SUPER^.InfoData.Diag.5 THEN
	Events.RaiseEvent(E_SafetyEstop.EDM2);
END_IF
END_METHOD

METHOD GetHighestActiveEventReaction : DINT
GetHighestActiveEventReaction := Events.GetHighestActiveEventReaction();
END_METHOD

METHOD GetHighestActiveEventSeverity : TcEventSeverity
GetHighestActiveEventSeverity := Events.GetHighestActiveEventSeverity();
END_METHOD

METHOD Reset
SUPER^.Reset();
Events.Reset();
END_METHOD

METHOD SetEventReactions
VAR_INPUT
	Verbose	 : DINT := 0;
	Info	 : DINT := 1;
	Warning	 : DINT := 2;
	Error	 : DINT := 3;
	Critical : DINT := 4;
END_VAR
Events.SetEventReactions(Verbose,
						 Info,
						 Warning,
						 Error,
						 Critical);
END_METHOD

{attribute 'monitoring' := 'call'}
PROPERTY ActiveName : STRING
SET
_ActiveName := ActiveName;
END_SET
END_PROPERTY

(*FB_Init is always available implicitly and it is used primarily for initialization.
The return value is not evaluated. For a specific influence, you can also declare the
methods explicitly and provide additional code there with the standard initialization
code. You can evaluate the return value.*)
METHOD FB_Init : BOOL
VAR_INPUT
	(* TRUE: the retain variables are initialized (reset warm / reset cold)*)
	bInitRetains : BOOL;

	(* TRUE: the instance will be copied to the copy code afterward (online change)   *)
	bInCopyCode : BOOL;
	Name		: T_MaxString;
END_VAR
Events.GenerateTcEvents(Name, ADR(TC_events.SafetyEstop), SIZEOF(ST_SafetyEstop));
END_METHOD

PROPERTY SafetyGroup : I_TaskResult
SET
_SafetyGroup := SafetyGroup;
END_SET
END_PROPERTY

END_FUNCTION_BLOCK

// Components/Safety/SafetyGroup_TcEvents
FUNCTION_BLOCK SafetyGroup_TcEvents EXTENDS SafetyBase IMPLEMENTS I_EventReactionTcEvents
VAR
	Run AT %Q* : BOOL;
	Events	   : TcEventClass('Safety Group Events');
	{attribute 'hide'}
	_AutoResetFaults : BOOL;
END_VAR

METHOD CyclicLogic
VAR_INST
	LinkErrorRun	 : BOOL;
	AutoFaultAck	 : TON;
	TriggerAutoReset : R_TRIG;
END_VAR
SUPER^.CyclicLogic();
IF NOT LinkErrorRun AND NOT Simulated AND (F_GetMappingStatus(ADR(Run), SIZEOF(Run)) = EplcMappingStatus.MS_Unmapped) THEN
	LinkErrorRun := TRUE;
	Trace.LogMessage(Name, 'Group Run not mapped to Safety!');
END_IF

Run := TRUE;
IF _ResetFunction <> 0 THEN
	AutoFaultAck(IN := (_AutoResetFaults AND (SUPER^.InfoData.Diag <> 0)) AND NOT _ResetFunction.Busy, PT := T#250MS);
	TriggerAutoReset(CLK := AutoFaultAck.Q);
	IF TriggerAutoReset.Q THEN
		_ResetFunction.Execute();
	END_IF

	_Busy := _ResetFunction.Busy;
END_IF

_OK	   := SUPER^.InfoData.State = E_SafetyGroup_State.Run;
_Error := GetHighestActiveEventReaction() >= TcEventSeverity.Error;
IF _ResetFunction <> 0 AND_THEN _ResetFunction.Busy THEN
	RETURN;
END_IF

IF SUPER^.InfoData.Diag = E_SafetyGroup_Diag.FbError THEN
	Events.RaiseEvent(E_SafetyGroup.FbError);
END_IF

IF SUPER^.InfoData.Diag = E_SafetyGroup_Diag.ComError THEN
	Events.RaiseEvent(E_SafetyGroup.ComError);
END_IF

IF SUPER^.InfoData.Diag = E_SafetyGroup_Diag.ModuleError THEN
	Events.RaiseEvent(E_SafetyGroup.ModuleError);
END_IF

IF SUPER^.InfoData.Diag = E_SafetyGroup_Diag.CmpError THEN
	Events.RaiseEvent(E_SafetyGroup.CmpError);
END_IF

IF SUPER^.InfoData.Diag = E_SafetyGroup_Diag.DeactiveError THEN
	Events.RaiseEvent(E_SafetyGroup.DeactiveError);
END_IF

IF SUPER^.InfoData.Diag = E_SafetyGroup_Diag.RestartError THEN
	Events.RaiseEvent(E_SafetyGroup.RestartError);
END_IF
END_METHOD

METHOD GetHighestActiveEventReaction : DINT
GetHighestActiveEventReaction := Events.GetHighestActiveEventReaction();
END_METHOD

METHOD GetHighestActiveEventSeverity : TcEventSeverity
GetHighestActiveEventSeverity := Events.GetHighestActiveEventSeverity();
END_METHOD

METHOD Reset
SUPER^.Reset();
Events.Reset();
END_METHOD

METHOD SetEventReactions
VAR_INPUT
	Verbose	 : DINT := 0;
	Info	 : DINT := 1;
	Warning	 : DINT := 2;
	Error	 : DINT := 3;
	Critical : DINT := 4;
END_VAR
Events.SetEventReactions(Verbose,
						 Info,
						 Warning,
						 Error,
						 Critical);
END_METHOD

{attribute 'monitoring' := 'call'}
PROPERTY AutoResetFaults : BOOL
GET
AutoResetFaults := _AutoResetFaults;
END_GET
SET
_AutoResetFaults := AutoResetFaults;
END_SET
END_PROPERTY

(*FB_Init is always available implicitly and it is used primarily for initialization.
The return value is not evaluated. For a specific influence, you can also declare the
methods explicitly and provide additional code there with the standard initialization
code. You can evaluate the return value.*)
METHOD FB_Init : BOOL
VAR_INPUT
	(* TRUE: the retain variables are initialized (reset warm / reset cold)*)
	bInitRetains : BOOL;

	(* TRUE: the instance will be copied to the copy code afterward (online change)   *)
	bInCopyCode : BOOL;
	Name		: T_MaxString;
END_VAR
Events.GenerateTcEvents(Name, ADR(TC_events.SafetyGroup), SIZEOF(ST_SafetyGroup));
END_METHOD

END_FUNCTION_BLOCK

// Components/Safety/SafetyModule
FUNCTION_BLOCK SafetyModule EXTENDS Module IMPLEMENTS I_SafetyModule
VAR
	SequenceState			 : UDINT;
	TwinSAFEResetDelay		 : TON;
	SafetyPLC_WcState AT %I* : BOOL;
	SafetyPLC_AmsAddr AT %I* : AMSADDR;
	_SafetyPlcCoE			 : CoeDevice('Safety PLC') := (AdsAddr := SafetyPLC_AmsAddr);
	_SafetyAddressInfo		 : ST_SafetyAddressInfo;
END_VAR

VAR
	GetComponentsTaskResultVisitor : GetComponentsTaskResultVisitor;
	SetSafetySimulationVisitor	   : SetSafetySimulationVisitor;
	SafetyOkVisitor				   : SafetyOkVisitor;
END_VAR

METHOD OnCyclicCall
IF NOT Initialized THEN
	Initialize();
	RETURN;
END_IF

TwinSAFEResetDelay(PT := T#250MS);
CASE SequenceState OF
	0:
		TwinSAFEResetDelay.IN := FALSE;

	10:
		ResetComponents();
		SequenceState := 20;

	20:
		TwinSAFEResetDelay.IN := TRUE;
		IF TwinSAFEResetDelay.Q THEN
			SequenceState := 0;
		END_IF
END_CASE

GetComponentsTaskResultVisitor.Update(THIS^);
SafetyOkVisitor.Check(Components);
END_METHOD

(* This Module will be done initialize when ModuleInitialized := TRUE;, subequently all subitems will be called to be initialized *)
METHOD Initializing
_SafetyPlcCoE.CyclicLogic();
CASE SequenceState OF
	0:
		IF F_GetMappingStatus(ADR(SafetyPLC_WcState), SIZEOF(SafetyPLC_WcState)) = EplcMappingStatus.MS_Unmapped OR F_GetMappingStatus(ADR(SafetyPLC_AmsAddr), SIZEOF(SafetyPLC_AmsAddr)) = EplcMappingStatus.MS_Unmapped THEN
			SequenceState := 100;
			Trace.LogMessage(Name, 'Safety PLC not mapped, info will not be read!');
		ELSE
			SequenceState := SequenceState + 10;
		END_IF

	10:
		IF NOT SafetyPLC_WcState THEN
			SequenceState := SequenceState + 10;
		END_IF

	20:
		SafetyPlcCoE.Read(16#F980,
						  1,
						  ADR(_SafetyAddressInfo.FSoEAddress),
						  SIZEOF(_SafetyAddressInfo.FSoEAddress));

		SequenceState := SequenceState + 1;

	21:
		IF NOT SafetyPlcCoE.Error AND NOT SafetyPlcCoE.Busy THEN
			SequenceState := SequenceState + 1;
		END_IF

	22:
		SafetyPlcCoE.Read(16#F980,
						  2,
						  ADR(_SafetyAddressInfo.SerialNumber),
						  SIZEOF(_SafetyAddressInfo.SerialNumber));

		SequenceState := SequenceState + 1;

	23:
		IF NOT SafetyPlcCoE.Error AND NOT SafetyPlcCoE.Busy THEN
			SequenceState := SequenceState + 1;
		END_IF

	24:
		SafetyPlcCoE.Read(16#F980,
						  3,
						  ADR(_SafetyAddressInfo.ProjectCRC),
						  SIZEOF(_SafetyAddressInfo.ProjectCRC));

		SequenceState := SequenceState + 1;

	25:
		IF NOT SafetyPlcCoE.Error AND NOT SafetyPlcCoE.Busy THEN
			SequenceState := SequenceState + 1;
		END_IF

	26:
		SafetyPlcCoE.Read(16#F980,
						  4,
						  ADR(_SafetyAddressInfo.DefaultProjectCRC),
						  SIZEOF(_SafetyAddressInfo.DefaultProjectCRC));

		SequenceState := SequenceState + 1;

	27:
		IF NOT SafetyPlcCoE.Error AND NOT SafetyPlcCoE.Busy THEN
			SequenceState := 100;
		END_IF

	100:
		SequenceState	  := 0;
		ModuleInitialized := TRUE;
END_CASE
END_METHOD

{attribute 'monitoring' := 'call'}
PROPERTY Simulated : BOOL
GET
Simulated := SetSafetySimulationVisitor.Simulated;
END_GET
SET
SetSafetySimulationVisitor.Simulated := Simulated;
Components.Accept(SetSafetySimulationVisitor);
END_SET
END_PROPERTY

METHOD SimulateSafetyDiag
VAR_INPUT
	SimulationValueDiag : UINT;
END_VAR
SetSafetySimulationVisitor.Diag := SimulationValueDiag;
Components.Accept(SetSafetySimulationVisitor);
END_METHOD

METHOD SimulateSafetyState
VAR_INPUT
	SimulationValueState : USINT;
END_VAR
SetSafetySimulationVisitor.State := SimulationValueState;
Components.Accept(SetSafetySimulationVisitor);
END_METHOD

{attribute 'monitoring' := 'call'}
PROPERTY Busy : BOOL
GET
Busy := SequenceState <> 0;
END_GET
END_PROPERTY

{attribute 'monitoring' := 'call'}
PROPERTY Error : BOOL
GET
Error := GetComponentsTaskResultVisitor.Error;
END_GET
END_PROPERTY

{attribute 'monitoring' := 'call'}
PROPERTY ErrorId : UDINT
GET
ErrorId := GetComponentsTaskResultVisitor.ErrorId;
END_GET
END_PROPERTY

METHOD AddSafetyComponent
VAR_INPUT
	Component : I_SafetyBase;
END_VAR
Component.RegisterWithParent(THIS^);
END_METHOD

(*FB_Init is always available implicitly and it is used primarily for initialization.
The return value is not evaluated. For a specific influence, you can also declare the
methods explicitly and provide additional code there with the standard initialization
code. You can evaluate the return value.*)
METHOD FB_Init : BOOL
VAR_INPUT
	(* TRUE: the retain variables are initialized (reset warm / reset cold)*)
	bInitRetains : BOOL;

	(* TRUE: the instance will be copied to the copy code afterward (online change)   *)
	bInCopyCode : BOOL;
	Name		: T_MaxString;
END_VAR
SafetyPlcCoE.RegisterWithParent(THIS^);
END_METHOD

{attribute 'monitoring' := 'call'}
PROPERTY OK : BOOL
GET
OK := SafetyOkVisitor.OK;
END_GET
END_PROPERTY

METHOD Reset
IF Busy THEN
	RETURN;
END_IF

SequenceState := 10;
END_METHOD

PROPERTY SafetyAddressInfo : REFERENCE TO ST_SafetyAddressInfo
GET
SafetyAddressInfo REF= _SafetyAddressInfo;
END_GET
END_PROPERTY

PROPERTY SafetyPlcCoE : I_CoeDevice
GET
SafetyPlcCoE := _SafetyPlcCoE;
END_GET
END_PROPERTY

END_FUNCTION_BLOCK

// Visitors/Reset/GetComponentsTaskResultVisitor
FUNCTION_BLOCK GetComponentsTaskResultVisitor IMPLEMENTS I_ComponentVisitor, I_TaskResult
VAR
	{attribute 'hide'}
	Result : I_TaskResult;
	{attribute 'hide'}
	_Busy : BOOL;
	{attribute 'hide'}
	_Error : BOOL;
	{attribute 'hide'}
	_ErrorId : UDINT;
END_VAR

{attribute 'monitoring' := 'call'}
PROPERTY Busy : BOOL
GET
Busy := _Busy;
END_GET
END_PROPERTY

{attribute 'monitoring' := 'call'}
PROPERTY Error : BOOL
GET
Error := _Error;
END_GET
END_PROPERTY

{attribute 'monitoring' := 'call'}
PROPERTY ErrorId : UDINT
GET
ErrorID := _ErrorID;
END_GET
END_PROPERTY

METHOD Update
VAR_INPUT
	Module : I_Module;
END_VAR
_Error	 := FALSE;
_ErrorId := 0;
_Busy	 := FALSE;
Module.Components.Accept(THIS^);
END_METHOD

METHOD VisitComponent
VAR_INPUT
	Component : I_Component;
END_VAR
IF __QUERYINTERFACE(Component, Result) THEN
	IF Result.Error THEN
		_Error	 := TRUE;
		_ErrorId := Result.ErrorId;
	END_IF

	IF Result.Busy THEN
		_Busy := TRUE;
	END_IF
END_IF
END_METHOD

END_FUNCTION_BLOCK

// Components/Safety/SafetyMonFB_TcEvents
FUNCTION_BLOCK SafetyMonFB_TcEvents EXTENDS SafetyBase IMPLEMENTS I_EventReactionTcEvents, I_InSafetyGroup
VAR
	{attribute 'hide'}
	_ActiveAlarm : BOOL := TRUE;
	{attribute 'hide'}
	_ActiveName	 : STRING := 'pressed!';
	Events		 : TcEventClass('Safety MonFB Events');
	_SafetyGroup : I_TaskResult;
END_VAR

METHOD CyclicLogic
SUPER^.CyclicLogic();
_OK	   := SUPER^.InfoData.State = E_SafetyMon_State.Run;
_Error := GetHighestActiveEventReaction() >= TcEventSeverity.Error;
IF _SafetyGroup <> 0 THEN
	IF _SafetyGroup.Error THEN
		Events.Reset();
		RETURN;
	END_IF
END_IF

IF _ResetFunction <> 0 AND_THEN _ResetFunction.Busy THEN
	RETURN;
END_IF

IF NOT SUPER^.OK AND _ActiveAlarm THEN
	Events.Arguments(E_SafetyMon.Active).Clear().AddString(_ActiveName);
	Events.RaiseEvent(E_SafetyMon.Active);
END_IF

IF SUPER^.InfoData.Diag.0 THEN
	Events.RaiseEvent(E_SafetyMon.Disc1);
END_IF

IF SUPER^.InfoData.Diag.1 THEN
	Events.RaiseEvent(E_SafetyMon.Disc2);
END_IF

IF SUPER^.InfoData.Diag.2 THEN
	Events.RaiseEvent(E_SafetyMon.DiscInput);
END_IF

IF SUPER^.InfoData.Diag.4 THEN
	Events.RaiseEvent(E_SafetyMon.Edm1);
END_IF

IF SUPER^.InfoData.Diag.5 THEN
	Events.RaiseEvent(E_SafetyMon.Edm2);
END_IF

IF SUPER^.InfoData.Diag.8 THEN
	Events.RaiseEvent(E_SafetyMon.Disc1Safe);
END_IF

IF SUPER^.InfoData.Diag.9 THEN
	Events.RaiseEvent(E_SafetyMon.Disc2Safe);
END_IF

IF SUPER^.InfoData.Diag.10 THEN
	Events.RaiseEvent(E_SafetyMon.DiscInputSafe);
END_IF
END_METHOD

METHOD GetHighestActiveEventReaction : DINT
GetHighestActiveEventReaction := Events.GetHighestActiveEventReaction();
END_METHOD

METHOD GetHighestActiveEventSeverity : TcEventSeverity
GetHighestActiveEventSeverity := Events.GetHighestActiveEventSeverity();
END_METHOD

METHOD Reset
SUPER^.Reset();
Events.Reset();
END_METHOD

METHOD SetEventReactions
VAR_INPUT
	Verbose	 : DINT := 0;
	Info	 : DINT := 1;
	Warning	 : DINT := 2;
	Error	 : DINT := 3;
	Critical : DINT := 4;
END_VAR
Events.SetEventReactions(Verbose,
						 Info,
						 Warning,
						 Error,
						 Critical);
END_METHOD

PROPERTY ActiveAlarm : BOOL
SET
_ActiveAlarm := ActiveAlarm;
END_SET
END_PROPERTY

PROPERTY ActiveName : STRING
SET
_ActiveName := ActiveName;
END_SET
END_PROPERTY

(*FB_Init is always available implicitly and it is used primarily for initialization.
The return value is not evaluated. For a specific influence, you can also declare the
methods explicitly and provide additional code there with the standard initialization
code. You can evaluate the return value.*)
METHOD FB_Init : BOOL
VAR_INPUT
	(* TRUE: the retain variables are initialized (reset warm / reset cold)*)
	bInitRetains : BOOL;

	(* TRUE: the instance will be copied to the copy code afterward (online change)   *)
	bInCopyCode : BOOL;
	Name		: T_MaxString;
END_VAR
Events.GenerateTcEvents(Name, ADR(TC_events.SafetyMon), SIZEOF(ST_SafetyMon));
END_METHOD

PROPERTY SafetyGroup : I_TaskResult
SET
_SafetyGroup := SafetyGroup;
END_SET
END_PROPERTY

END_FUNCTION_BLOCK

// Components/Serial/Interface/I_SerialByteConnection
INTERFACE I_SerialByteConnection

PROPERTY ByteData : BYTE
GET
END_GET
END_PROPERTY

PROPERTY ByteDataRecieved : BOOL
GET
END_GET
END_PROPERTY

METHOD SendAByte : HRESULT
VAR_INPUT
	DataToSend : BYTE;
END_VAR
END_METHOD

END_INTERFACE

// Components/Serial/Interface/I_SerialLineControl
INTERFACE I_SerialLineControl EXTENDS I_Cyclic

PROPERTY rxBuffer : REFERENCE TO combuffer
GET
END_GET
END_PROPERTY

PROPERTY txBuffer : REFERENCE TO combuffer
GET
END_GET
END_PROPERTY

END_INTERFACE

// Components/Serial/Interface/I_SerialStringConnection
INTERFACE I_SerialStringConnection

METHOD SendAString : HRESULT
VAR_INPUT
	DataToSend : T_MaxString;
END_VAR
END_METHOD

PROPERTY StringData : t_maxstring
GET
END_GET
END_PROPERTY

PROPERTY StringRecieved : BOOL
GET
END_GET
END_PROPERTY

END_INTERFACE

// Components/Serial/SerialByteConnection
FUNCTION_BLOCK SerialByteConnection EXTENDS CyclicComponent IMPLEMENTS I_SerialByteConnection
VAR
	sendSerialByte		: SendByte;
	recieveSerialByte	: ReceiveByte;
	clearTheComBuffer	: ClearComBuffer;
	MySerialLineControl : I_SerialLineControl;
	_ByteDataRecieved	: BYTE;
	_RecieveError		: ComError_t;
	_SendError			: ComError_t;
	RecieveCounter		: UDINT;
	_ByteRecieved		: BOOL;
END_VAR

PROPERTY ByteData : Byte
GET
ByteData := _ByteDataRecieved;
END_GET
END_PROPERTY

PROPERTY ByteDataRecieved : BOOL
GET
ByteDataRecieved := _ByteRecieved;
_ByteRecieved := FALSE;
END_GET
END_PROPERTY

METHOD CyclicLogic
IF MySerialLineControl = 0 THEN
	RETURN;
END_IF

IF recieveSerialByte.ByteReceived THEN
	_ByteDataRecieved := recieveSerialByte.ReceivedByte;
	RecieveCounter	  := RecieveCounter + 1;
	_ByteRecieved	  := TRUE;
END_IF

recieveSerialByte(Error => _RecieveError, RxBuffer := MySerialLineControl.rxBuffer);
END_METHOD

//FB_Init is always available implicitly and it is used primarily for initialization.

//The return value is not evaluated. For a specific influence, you can also declare the

//methods explicitly and provide additional code there with the standard initialization

//code. You can evaluate the return value.
METHOD FB_Init : BOOL
VAR_INPUT
	bInitRetains		 : BOOL; // TRUE: the retain variables are initialized (reset warm / reset cold)
	bInCopyCode			 : BOOL; // TRUE: the instance will be copied to the copy code afterward (online change)   
	Name				 : T_MaxString;
	SerialLineController : I_SerialLineControl;
END_VAR
SetDependencies(SerialLineController);
END_METHOD

METHOD Reset : HRESULT;
VAR_INPUT
END_VAR
IF MySerialLineControl = 0 THEN
	Reset := -1;
	trace.Error(Source := 'SerialConnection', 'No LineControl for Sending');
	RETURN;
END_IF

clearTheComBuffer(Buffer := MySerialLineControl.rxBuffer);
_ByteDataRecieved := 0;
_ByteRecieved	  := FALSE;
RecieveCounter	  := 0;
END_METHOD

METHOD SendAByte : HRESULT
VAR_INPUT
	DataToSend : BYTE;
END_VAR
IF MySerialLineControl = 0 THEN
	SendAByte := -1;
	trace.Error(Source := 'SerialConnection', 'No LineControl for Sending');
	RETURN;
END_IF

sendSerialByte(SendByte := DataToSend, Error => _SendError, TxBuffer := MySerialLineControl.txBuffer);
END_METHOD

METHOD SetDependencies : BOOL
VAR_INPUT
	SerialLineController : I_SerialLineControl;
END_VAR
IF SerialLineController = 0 THEN
	RETURN;
END_IF

MySerialLineControl := SerialLineController;
SetDependencies		:= TRUE;
END_METHOD

END_FUNCTION_BLOCK

// Components/Serial/SerialLineControl_ADS
FUNCTION_BLOCK SerialLineControl_ADS IMPLEMENTS I_Cyclic, I_SerialLineControl
VAR
	seriallinectrl : SerialLineControlADS := (Timeout := T#5S);
	txComBuffer	   : Tc2_SerialCom.ComBuffer;
	rxComBuffer	   : Tc2_SerialCom.ComBuffer;
END_VAR

METHOD CyclicLogic
seriallinectrl(Connect := TRUE, TxBuffer := txComBuffer, RxBuffer := rxComBuffer);
END_METHOD

PROPERTY rxBuffer : REFERENCE TO combuffer
GET
rxBuffer REF= rxComBuffer;
END_GET
END_PROPERTY

METHOD SetConnectionConfig : BOOL
VAR_INPUT
	ComportSettings : ComSerialConfig;
	NetId			: T_AmsNetId := '';
END_VAR
seriallinectrl.SerialCfg := ComportSettings;
seriallinectrl.NetId	 := NetId;
SetConnectionConfig		 := TRUE;
END_METHOD

PROPERTY txBuffer : REFERENCE TO combuffer
GET
txBuffer REF= txComBuffer;
END_GET
END_PROPERTY

END_FUNCTION_BLOCK

// Components/Serial/SerialLineControl_Terminal
FUNCTION_BLOCK SerialLineControl_Terminal IMPLEMENTS I_Cyclic, I_SerialLineControl
VAR
	SerialLineCtrl : SerialLineControl;
	_serialMode	   : ComSerialLineMode_t := ComSerialLineMode_t.SERIALLINEMODE_EL6_22B;
	txComBuffer	   : Tc2_SerialCom.ComBuffer;
	rxComBuffer	   : Tc2_SerialCom.ComBuffer;
	_ComIn		   : POINTER TO ARRAY[0..65] OF BYTE;
	_ComOut		   : POINTER TO ARRAY[0..65] OF BYTE;
	_SizeComIn	   : INT;
END_VAR

METHOD CyclicLogic
IF _ComIn = 0 OR _ComOut = 0 THEN
	RETURN;
END_IF

SerialLineCtrl(Mode		 := _serialMode,
			   pComIn	 := _ComIn,
			   pComOut	 := _ComOut,
			   SizeComIn := _SizeComIn,
			   TxBuffer	 := txComBuffer,
			   RxBuffer	 := rxComBuffer);
END_METHOD

//FB_Init is always available implicitly and it is used primarily for initialization.

//The return value is not evaluated. For a specific influence, you can also declare the

//methods explicitly and provide additional code there with the standard initialization

//code. You can evaluate the return value.
METHOD FB_Init : BOOL
VAR_INPUT
	bInitRetains : BOOL; // TRUE: the retain variables are initialized (reset warm / reset cold)
	bInCopyCode	 : BOOL; // TRUE: the instance will be copied to the copy code afterward (online change)   
	ComIn		 : POINTER TO ARRAY[0..65] OF BYTE;
	ComOut		 : POINTER TO ARRAY[0..65] OF BYTE;
END_VAR
SetDependencies(ComIn, ComOut);
END_METHOD

PROPERTY rxBuffer : REFERENCE TO combuffer
GET
rxBuffer REF= rxComBuffer;
END_GET
END_PROPERTY

METHOD SetConnectionConfig : BOOL
VAR_INPUT
	SizeComIn  : INT;
	SerialMode : ComSerialLineMode_t;
END_VAR
_SizeComIn	:= SizeComIn;
_serialMode := SerialMode;
END_METHOD

METHOD SetDependencies : BOOL
VAR_INPUT
	ComIn  : POINTER TO ARRAY[0..65] OF BYTE;
	ComOut : POINTER TO ARRAY[0..65] OF BYTE;
END_VAR
_ComIn	:= ComIn;
_ComOut := ComOut;
END_METHOD

PROPERTY txBuffer : REFERENCE TO combuffer
GET
txBuffer REF= txComBuffer;
END_GET
END_PROPERTY

END_FUNCTION_BLOCK

// Components/Serial/SerialStringConnection
FUNCTION_BLOCK SerialStringConnection EXTENDS CyclicComponent IMPLEMENTS I_SerialStringConnection
VAR
	sendSerialString	: SendString255;
	receiveSerialString : ReceiveString255;
	clearTheComBuffer	: ClearComBuffer;
	MySerialLineControl : I_SerialLineControl;
	_StringDataRecieved : T_MaxString;
	_RecieveError		: ComError_t;
	_SendError			: ComError_t;
	RecieveCounter		: UDINT;
	_StringReceived		: BOOL;
END_VAR

METHOD CyclicLogic
IF MySerialLineControl = 0 THEN
	RETURN;
END_IF

IF receiveSerialString.StringReceived THEN
	_StringReceived := TRUE;
	RecieveCounter	:= RecieveCounter + 1;
END_IF

receiveSerialString(ReceivedString := _StringDataRecieved, Error => _RecieveError, RXbuffer := MySerialLineControl.rxBuffer);
END_METHOD

//FB_Init is always available implicitly and it is used primarily for initialization.

//The return value is not evaluated. For a specific influence, you can also declare the

//methods explicitly and provide additional code there with the standard initialization

//code. You can evaluate the return value.
METHOD FB_Init : BOOL
VAR_INPUT
	bInitRetains		 : BOOL; // TRUE: the retain variables are initialized (reset warm / reset cold)
	bInCopyCode			 : BOOL; // TRUE: the instance will be copied to the copy code afterward (online change)   
	Name				 : T_MaxString;
	SerialLineController : I_SerialLineControl;
END_VAR
SetDependencies(SerialLineController);
END_METHOD

METHOD Reset : HRESULT
VAR_INPUT
END_VAR
IF MySerialLineControl = 0 THEN
	Reset := -1;
	trace.Error(Source := 'SerialConnection', 'No LineControl for Sending');
	RETURN;
END_IF

clearTheComBuffer(Buffer := MySerialLineControl.rxBuffer);
_StringDataRecieved := '';
_StringReceived		:= FALSE;
RecieveCounter		:= 0;
END_METHOD

METHOD SendAString : HRESULT
VAR_INPUT
	DataToSend : T_MaxString;
END_VAR
IF MySerialLineControl = 0 THEN
	SendAString := -1;
	trace.Error(Source := 'SerialConnection', 'No LineControl for Sending');
	RETURN;
END_IF

sendSerialString(SendString := DataToSend, Error => _SendError, TXbuffer := MySerialLineControl.txBuffer);
END_METHOD

METHOD SetDependencies : BOOL
VAR_INPUT
	SerialLineController : I_SerialLineControl;
END_VAR
IF SerialLineController = 0 THEN
	RETURN;
END_IF

MySerialLineControl := SerialLineController;
SetDependencies		:= TRUE;
END_METHOD

METHOD SetSerialConfiguration : BOOL
VAR_INPUT
	Prefix : STRING;
	Suffix : STRING;
END_VAR
receiveSerialString.Prefix := Prefix;
receiveSerialString.Suffix := Suffix;
END_METHOD

PROPERTY StringData : t_maxstring
GET
StringData := _StringDataRecieved;
END_GET
END_PROPERTY

PROPERTY StringRecieved : BOOL
GET
StringRecieved	:= _StringReceived;
_StringReceived := FALSE;
END_GET
END_PROPERTY

END_FUNCTION_BLOCK

// Components/Tcp Ip/Interface/I_TcpIpConnection
INTERFACE I_TcpIpConnection EXTENDS I_Component

{attribute 'monitoring' := 'call'}
PROPERTY ConnectionState : E_SocketConnectionState
GET
END_GET
END_PROPERTY

{attribute 'monitoring' := 'call'}
PROPERTY IP : T_IPv4Addr
SET
END_SET
END_PROPERTY

{attribute 'monitoring' := 'call'}
PROPERTY Port : UDINT
SET
END_SET
END_PROPERTY

METHOD RegisterCommand
VAR_INPUT
	Command : I_TcpIpSubscription;
END_VAR
END_METHOD

METHOD SendCommand
VAR_INPUT
	Command : POINTER TO ST_TcpIpPayload;
END_VAR
END_METHOD

METHOD SendPriorityCommand
VAR_INPUT
	Command : POINTER TO ST_TcpIpPayload;
END_VAR
END_METHOD

PROPERTY Socket : T_HSOCKET
GET
END_GET
END_PROPERTY

END_INTERFACE

// Components/Tcp Ip/Interface/I_TcpIpSubscription
INTERFACE I_TcpIpSubscription EXTENDS I_Base

METHOD UpdateCommandResult
VAR_INPUT
	Response : POINTER TO ST_TcpIpPayload;
END_VAR
END_METHOD

END_INTERFACE

// Components/Tcp Ip/TcpIpCommandResultFilter
FUNCTION_BLOCK ABSTRACT TcpIpCommandResultFilter EXTENDS CyclicComponent IMPLEMENTS I_TcpIpSubscription
VAR
	TcpIpConnection : I_TcpIpConnection;
	{attribute 'hide'}
	_Initialized   : BOOL := FALSE;
	CommandActive  : BOOL;
	CommandTimeout : TON;
END_VAR

METHOD CyclicLogic
CommandTimeout(IN := CommandActive, PT := T#10S);
IF CommandTimeout.Q THEN
	CommandActive := FALSE;
	Trace.Info(_Name, CONCAT('Command response not recieved! ', Name));
END_IF
END_METHOD

(*FB_Init is always available implicitly and it is used primarily for initialization.
The return value is not evaluated. For a specific influence, you can also declare the
methods explicitly and provide additional code there with the standard initialization
code. You can evaluate the return value.*)
METHOD FB_Init : BOOL
VAR_INPUT
	(* TRUE: the retain variables are initialized (reset warm / reset cold)*)
	bInitRetains : BOOL;

	(* TRUE: the instance will be copied to the copy code afterward (online change)   *)
	bInCopyCode		: BOOL;
	Name			: T_MaxString;
	TcpIpConnection : I_TcpIpConnection;
END_VAR
THIS^.TcpIpConnection := TcpIpConnection;
TcpIpConnection.RegisterCommand(THIS^);
END_METHOD

METHOD ABSTRACT UpdateCommandResult
VAR_INPUT
	Response : POINTER TO ST_TcpIpPayload;
END_VAR
// Filter incoming TcpIp traffic here!
END_METHOD

END_FUNCTION_BLOCK

// Components/Tcp Ip/TcpIpConnection
FUNCTION_BLOCK TcpIpConnection EXTENDS CyclicComponent IMPLEMENTS I_TcpIpConnection, I_Initializable
VAR
	_Initialized   : BOOL;
	_IP			   : T_IPv4Addr := '127.0.0.1';
	_Port		   : UDINT;
	SocketCloseAll : FB_SocketCloseAll;

